# B&R Automation Studio project MappAssetInt
Automation Studio 4.12.6.106; technology packages: mapp 5.24.2

## Configuration X20CP

CPU X20CP3687X, AutomationRuntime J4.93, Build 4.1.2, Safety 0.0, Vc V4.73.3

### Task classes (Cpu.sw)
```
Cyclic#8:
  AssetTest <- AssetTest.prg
  Sample <- exAssetInt.Sample.prg
  Shift <- Shift.prg
VcDataObjects: Vis <- Vis.dob
Binaries: vcnet, udbdef, vcrt, vcpkat, vcctext, vctcal, vcfile, vcgclass, vccstr, vcpdsw, arial, vcdsint, vcmgr, vcdsloc, vcfntttf, vccovl, vcshared, arialbd, vcalarm, vccdt, vcpdvnc, vcpfar00, vcbclass, TCData, vccnum, arsvcreg, vccshape, vccbtn, vccddbox, Vis01, Vis02, Vis03, vcclbox, vccpopup, arconfig, User, Config, ashwd, ashwac, Role, asfw, iomap, sysconf, vcpfx20, Visu01, Visu03, Visu02, Config_1
Libraries: AsBrStr, MpData, MpBase, MpAssetInt, MpCom, FileIO, DataObj, astime, brsystem, sys_lib, runtime, standard, vcresman, asieccon, ashw, AsIODiag, exAssetInt
```

### Hardware
```
X20CP3687X : X20CP3687X v1.8.0.0
  Connector IF2:
    ActivateDevice = 1
    Vnc1
    VncVcObjectName1 = Vis
    VncKeyMappingFile1 = VC\PS2-Keyboard.dis
    VncRefreshRate1 = 500
    ActivateSnmp = 2
  Connector IF3:
    DNAConfiguration = manual
    CycleTime = 2000
  ConfigurationID = MappAssetInt_X20CP1583
  UserPartitionSize = 16
  Simulation = 1
  UserRamSize = 731936
  RemMemSize = 300000
  TimerDeviceType = EPLX2X
  TimerDevice = X20CP3687X.IF3
  TaskClassIdleTime = 2000
  Cyclic1Duration = 2000
  Cyclic8Stack = 20000
  FileDevice1
  FileDeviceName1 = ARsim
  FileDevicePath1 = C:\Temp\AssetInt
  FileDevice2
  FileDeviceName2 = USER_HD
  FileDevicePath2 = F:\
  FtpUser1
  FtpUsername1 = admin
  FtpUserPassword1 = WA9hSMBXiqkZliudaf2dLB8I5WaEURjKd6F9iexMfBQ=
  FtpUserSalt1 = wS51ak4d
  FTPAccessRight1 = 0
  ActivateOpcUa = 1
  OpcUaInformationModels_PV_Version = 1
```

### Config.mpassetintcore - X20CP3687X/mappServices/Config.mpassetintcore
```
Element gAssetIntCore (Type=mpassetintcore)
  AssetInt:
    Shifts:
      [0]:
        Name = Morning
        TotalTime:
          Start = 21600000
          End = 50400000
        ScheduledDowntime:
          [0]:
            Reason = Lunch
            Start = 21780000
            End = 21900000
      [1]:
        Name = Afternoon
        TotalTime:
          Start = 50400000
          End = 79200000
        ScheduledDowntime:
          [0]:
            Reason = Dinner
            Start = 64800000
            End = 66600000
      [2]:
        Name = Night
        TotalTime:
          Start = 79200000
          End = 21600000
    Export:
      ColumnSeparator = ;
      DecimalMark = ,
  Alarms = MpAlarmX
```

## Configuration X20CP1583

CPU X20CP3586, AutomationRuntime I4.93, Build 4.1.2, Safety 0.0, Vc V4.73.1

CPU X20CP3687X, AutomationRuntime I4.93, Build 4.1.2, Safety 0.0, Vc V4.73.1

### Task classes (Cpu.sw)
```
Cyclic#4:
  AssetTest <- AssetTest.prg
Cyclic#8:
  Sample <- exAssetInt.Sample.prg
  Shift <- Shift.prg
VcDataObjects: Visu_R <- Visu_Resized.dob
Binaries: vcnet, udbdef, vcrt, vcpkat, vcctext, Visu01, vctcal, Visu03, vcfile, vcgclass, vccstr, vcpdsw, arial, vcdsint, vcmgr, vcdsloc, vcfntttf, Visu02, vccovl, vcshared, arialbd, vcalarm, vccdt, vcpdvnc, vcpfar00, vcbclass, TCData, vccnum, arsvcreg, vccshape, vccbtn, arconfig, User, Config, ashwd, ashwac, Role, asfw, iomap, sysconf, vcpfx20, Config_1
Libraries: AsBrStr, MpData, MpBase, MpAssetInt, MpCom, FileIO, DataObj, astime, brsystem, sys_lib, runtime, exAssetInt, vcresman, asieccon, ashw, standard
```

### Hardware
```
X20CP3687X : X20CP3687X v1.8.0.0
  Connector IF2:
    ActivateDevice = 1
    Vnc1
    VncVcObjectName1 = Vis
    VncKeyMappingFile1 = VC\PS2-Keyboard.dis
    VncRefreshRate1 = 500
    ActivateSnmp = 2
  Connector IF3:
    DNAConfiguration = manual
    CycleTime = 2000
  ConfigurationID = MappAssetInt_X20CP1583
  UserPartitionSize = 16
  UserRamSize = 731936
  RemMemSize = 300000
  Cyclic8Stack = 20000
  FileDevice1
  FileDeviceName1 = ARsim
  FileDevicePath1 = c:\Temp\AssetInt
  FileDevice2
  FileDeviceName2 = USER_HD
  FileDevicePath2 = f:\
  FtpUser1
  FtpUsername1 = admin
  FtpUserPassword1 = WA9hSMBXiqkZliudaf2dLB8I5WaEURjKd6F9iexMfBQ=
  FtpUserSalt1 = wS51ak4d
  FTPAccessRight1 = 0
```

### Config.mpassetintcore - X20CP3586/mappServices/Config.mpassetintcore
```
Element gAssetIntCore (Type=mpassetintcore)
  AssetInt:
    Shifts:
      [0]:
        Name = Morning
        TotalTime:
          Start = 21600000
          End = 50400000
        ScheduledDowntime:
          [0]:
            Reason = Lunch
            Start = 39600000
            End = 41400000
      [1]:
        Name = Afternoon
        TotalTime:
          Start = 50400000
          End = 79200000
        ScheduledDowntime:
          [0]:
            Reason = Dinner
            Start = 64800000
            End = 66600000
      [2]:
        Name = Night
        TotalTime:
          Start = 79200000
          End = 21600000
    Export:
      ColumnSeparator = ;
      DecimalMark = ,
  Alarms = MpAlarmX
```

### Config_1.mpdatarecorder - X20CP3586/mappServices/Config_1.mpdatarecorder
```
Element gDataRecorder (Type=mpdatarecorder)
  DataRecorder:
    MaxFileSize = 2000
    SaveInterval = 3600000
    BufferSize = 70
    TimeStampPattern = %Y %m %d %H:%M:%S
    AutoSave = FALSE
    OverwriteOldestFile = TRUE
  Alarms = MpAlarmX
```

## Configuration X20EM

CPU X20EM0612, AutomationRuntime J4.93, Build 4.1.2, Safety 0.0, Vc V4.73.2

### Task classes (Cpu.sw)
```
Cyclic#8:
  AssetTest <- AssetTest.prg
  Sample <- exAssetInt.Sample.prg
  Shift <- Shift.prg
VcDataObjects: Vis <- Vis.dob
Binaries: vcnet, udbdef, vcrt, vcpkat, vcctext, vctcal, vcfile, vcgclass, vccstr, vcpdsw, arial, vcdsint, vcmgr, vcdsloc, vcfntttf, vccovl, vcshared, arialbd, vcalarm, vccdt, vcpdvnc, vcpfar00, vcbclass, TCData, vccnum, arsvcreg, vccshape, vccbtn, vccddbox, Vis01, Vis02, Vis03, vcclbox, vccpopup, arconfig, User, Config, ashwd, ashwac, Role, asfw, iomap, sysconf, vcpfx20, Visu01, Visu03, Visu02, Config_1
Libraries: AsBrStr, MpData, MpBase, MpAssetInt, MpCom, FileIO, DataObj, astime, brsystem, sys_lib, runtime, exAssetInt, standard, vcresman, asieccon, ashw, AsIODiag
```

### Hardware
```
X20EM0612 : X20EM0612 v1.1.1.0
  Connector IF2:
    ActivateDevice = 1
    Vnc1
    VncVcObjectName1 = Visu
    VncKeyMappingFile1 = VC\PS2-Keyboard.dis
    VncRefreshRate1 = 500
    ActivateSnmp = 2
  Connector IF3:
    DNAConfiguration = manual
  ConfigurationID = MappAssetInt_X20CP1583
  UserPartitionSize = 16
  UserRamSize = 32000
  RemMemSize = 32000
  TimerDeviceType = EPLX2X
  TimerDevice = X20EM0612.IF3
  TaskClassIdleTime = 2000
  Cyclic1Duration = 2000
  Cyclic8Stack = 20000
  FileDevice1
  FileDeviceName1 = ARsim
  FileDevicePath1 = c:\Temp\AssetInt
  FileDevice2
  FileDeviceName2 = USER_HD
  FileDevicePath2 = f:\
  FtpUser1
  FtpUsername1 = admin
  FtpUserPassword1 = WA9hSMBXiqkZliudaf2dLB8I5WaEURjKd6F9iexMfBQ=
  FtpUserSalt1 = wS51ak4d
  FTPAccessRight1 = 0
  ActivateOpcUa = 1
  OpcUaInformationModels_PV_Version = 1
```

### Config.mpassetintcore - X20EM0612/mappServices/Config.mpassetintcore
```
Element gAssetIntCore (Type=mpassetintcore)
  AssetInt:
    RecordingSizeShiftStatistics = 8
    RecordingSizeTimeline = 8
    RecordingSizeJobStatistics = 8
    Shifts:
      [0]:
        Name = Morning
        TotalTime:
          Start = 21600000
          End = 50400000
        ScheduledDowntime:
          [0]:
            Reason = Lunch
            Start = 21780000
            End = 21900000
      [1]:
        Name = Afternoon
        TotalTime:
          Start = 50400000
          End = 79200000
        ScheduledDowntime:
          [0]:
            Reason = Dinner
            Start = 64800000
            End = 66600000
      [2]:
        Name = Night
        TotalTime:
          Start = 79200000
          End = 21600000
    Export:
      ColumnSeparator = ;
      DecimalMark = ,
  Alarms = MpAlarmX
```

## Logical view

Binary libraries used (declarations not repeated): operator, runtime, astime, AsIecCon, sys_lib, DataObj, brsystem, FileIO, AsBrStr, standard, AsIODiag, MpAssetInt 5.24.2

### Global.typ - Globale Datentypen
```iecst
TYPE
	TIME_typ : 	STRUCT
		Hour : UDINT;
		Minutes : UDINT;
	END_STRUCT;
	SHIFT_typ : 	STRUCT
		Start : TIME_typ;
		End : TIME_typ;
		Name : STRING[20];
		ScheduledDowntime : ARRAY[0..9]OF DOWNTIME_typ;
	END_STRUCT;
	DOWNTIME_typ : 	STRUCT
		Start : TIME_typ;
		End : TIME_typ;
		Reason : STRING[20];
	END_STRUCT;
END_TYPE
```

### Global.var - Globale Variablen
```iecst
(*.-.-.-.-.---------------------------------------------------------------------------------------------------------------------------------------------------------------------------------*)
VAR
	gShift : ARRAY[0..4] OF SHIFT_typ;
	gAdditionalData : STRING[255] := 'Choclate';
	gNominalProductionRate : REAL := 3600;
	gDeviceName : STRING[50];
	gPieceCounterJob : UDINT;
	gPieceCounter : UDINT;
	gRejectCounter : UDINT;
	gRejectCounterRatio : UDINT := 10;
	gCurrentUser : STRING[50] := 'TylerDurden';
	gJobName : STRING[20] := 'Cookies';
	gDowntimeReason : STRING[50] := 'Winder is broken';
	gDowntime : exAssetIntDowntimeEnum;
	gCommandUpdate : BOOL;
	gCommandReset : BOOL;
	gCommandExport : BOOL;
	gCommandResetError : BOOL;
	gEnable : BOOL := TRUE;
	gLocked : UINT := 0;
END_VAR
```


### Program Logical/Shift (IEC)

#### Cyclic.st - Cyclic code
```iecst
PROGRAM _CYCLIC

	AssetIntPar.NominalProductionRate := gNominalProductionRate;
	AssetIntPar.AdditionalData := gAdditionalData;
	AssetIntPar.CurrentUser := gCurrentUser;
	AssetIntPar.Job := gJobName;

	MpAssetIntCore_0.PieceCounter := gPieceCounter;
	MpAssetIntCore_0.RejectCounter := gRejectCounter;

    MpAssetIntCore_0.MpLink := ADR(gAssetIntCore);
    MpAssetIntCore_0.Enable := gEnable;
    MpAssetIntCore_0.Parameters := ADR(AssetIntPar);
	MpAssetIntCore_0.DeviceName := ADR(gDeviceName);
	MpAssetIntCore_0.DowntimeReason := ADR(gDowntimeReason);
	MpAssetIntCore_0.Downtime := UDINT_TO_UINT(gDowntime);
	MpAssetIntCore_0.Update := gCommandUpdate;
	MpAssetIntCore_0.Reset := gCommandReset;
	MpAssetIntCore_0.Export := gCommandExport;
	MpAssetIntCore_0();

	IF EDGEPOS(MpAssetIntCore_0.UpdateDone) THEN
		gCommandUpdate := FALSE;
	END_IF

	AssetIntConfig.Export.DecimalMark := ',';
	AssetIntConfig.Export.ColumnSeparator := ';';
    brsstrcpy(ADR(AssetIntConfig.Export.JobStatisticsFileNamePattern), ADR('1234JobStatistics_%Y_%m_%d_%H_%M.csv'));
    brsstrcpy(ADR(AssetIntConfig.Export.ShiftStatisticsFileNamePattern), ADR('1234ShiftStatistics_%Y_%m_%d_%H_%M.csv'));
    brsstrcpy(ADR(AssetIntConfig.Export.TimelineFileNamePattern), ADR('1234Timeline_%Y_%m_%d_%H_%M.csv'));

	// --------------------------------------------------------------------------------------------------------------------------
	// Asset configuration
	FOR x := 0 TO SIZEOF(AssetIntConfig.Shifts)/SIZEOF(AssetIntConfig.Shifts[0]) - 1 DO
		AssetIntConfig.Shifts[x].Name := gShift[x].Name;
		FOR y := 0 TO SIZEOF(AssetIntConfig.Shifts[x].ScheduledDowntime)/SIZEOF(AssetIntConfig.Shifts[x].ScheduledDowntime[0]) - 1 DO
			AssetIntConfig.Shifts[x].ScheduledDowntime[y].Reason := gShift[x].ScheduledDowntime[y].Reason;
			AssetIntConfig.Shifts[x].ScheduledDowntime[y].Start := UDINT_TO_TOD((gShift[x].ScheduledDowntime[y].Start.Hour * 3600000) + (gShift[x].ScheduledDowntime[y].Start.Minutes * 60000));
			AssetIntConfig.Shifts[x].ScheduledDowntime[y].End := UDINT_TO_TOD((gShift[x].ScheduledDowntime[y].End.Hour * 3600000) + (gShift[x].ScheduledDowntime[y].End.Minutes * 60000));
		END_FOR;
		AssetIntConfig.Shifts[x].TotalTime.Start := UDINT_TO_TOD((gShift[x].Start.Hour * 3600000) + (gShift[x].Start.Minutes * 60000));
		AssetIntConfig.Shifts[x].TotalTime.End := UDINT_TO_TOD((gShift[x].End.Hour * 3600000) + (gShift[x].End.Minutes * 60000));
	END_FOR;

	IF (AssetIntConfig.Shifts[1].TotalTime.Start = AssetIntConfig.Shifts[0].TotalTime.End) AND (AssetIntConfig.Shifts[1].TotalTime.End <> AssetIntConfig.Shifts[1].TotalTime.Start) THEN
		AssetIntConfig.Shifts[1].TotalTime.Start := UDINT_TO_TOD((gShift[1].Start.Hour * 3600000) + (gShift[1].Start.Minutes * 60000) + 1);
	END_IF

	IF (AssetIntConfig.Shifts[2].TotalTime.Start = AssetIntConfig.Shifts[1].TotalTime.End) AND (AssetIntConfig.Shifts[2].TotalTime.End <> AssetIntConfig.Shifts[2].TotalTime.Start)  THEN
		AssetIntConfig.Shifts[2].TotalTime.Start := UDINT_TO_TOD((gShift[2].Start.Hour * 3600000) + (gShift[2].Start.Minutes * 60000) + 1);
	END_IF

	IF (AssetIntConfig.Shifts[0].TotalTime.Start = AssetIntConfig.Shifts[2].TotalTime.End) THEN
		AssetIntConfig.Shifts[0].TotalTime.Start := UDINT_TO_TOD((gShift[0].Start.Hour * 3600000) + (gShift[0].Start.Minutes * 60000) + 1);
	END_IF

    IF (AssetIntConfig.Shifts[1].TotalTime.Start = AssetIntConfig.Shifts[0].TotalTime.End) AND (AssetIntConfig.Shifts[1].TotalTime.End <> AssetIntConfig.Shifts[1].TotalTime.Start) THEN
        AssetIntConfig.Shifts[1].TotalTime.Start := UDINT_TO_TOD((gShift[1].Start.Hour * 3600000) + (gShift[1].Start.Minutes * 60000) + 1);
    END_IF

    IF (AssetIntConfig.Shifts[2].TotalTime.Start = AssetIntConfig.Shifts[1].TotalTime.End) AND (AssetIntConfig.Shifts[2].TotalTime.End <> AssetIntConfig.Shifts[2].TotalTime.Start)  THEN
        AssetIntConfig.Shifts[2].TotalTime.Start := UDINT_TO_TOD((gShift[2].Start.Hour * 3600000) + (gShift[2].Start.Minutes * 60000) + 1);
    END_IF

    IF (AssetIntConfig.Shifts[0].TotalTime.Start = AssetIntConfig.Shifts[2].TotalTime.End) THEN
        AssetIntConfig.Shifts[0].TotalTime.Start := UDINT_TO_TOD((gShift[0].Start.Hour * 3600000) + (gShift[0].Start.Minutes * 60000) + 1);
    END_IF

    IF (MpAssetIntCoreConfig_0.Save = 1) AND (MpAssetIntCoreConfig_0.CommandDone = 1) AND (MpAssetIntCoreConfig_0.CommandBusy = 0) THEN
        MpAssetIntCoreConfig_0.Save := 0;
    END_IF

    MpAssetIntCoreConfig_0.MpLink :=  ADR(gAssetIntCore);
    MpAssetIntCoreConfig_0.Enable := MpAssetIntCore_0.Active AND NOT DisableConfig;
    MpAssetIntCoreConfig_0.Configuration := ADR(AssetIntConfig);
    MpAssetIntCoreConfig_0();

    MpAssetIntShiftListUI_0.MpLink :=  ADR(gAssetIntCore);
    MpAssetIntShiftListUI_0.Enable := MpAssetIntCore_0.Active;
    MpAssetIntShiftListUI_0.UIConnect := ADR(ShiftListUIConnect);
	MpAssetIntShiftListUI_0.UISetup := ShiftListUISetup;
	MpAssetIntShiftListUI_0();

    MpAssetIntJobListUI_0.MpLink :=  ADR(gAssetIntCore);
    MpAssetIntJobListUI_0.Enable := MpAssetIntCore_0.Active;
	MpAssetIntJobListUI_0.UIConnect := ADR(JobListUIConnect);
	MpAssetIntJobListUI_0.UISetup := JobListUISetup;
	MpAssetIntJobListUI_0();

	MpAssetIntTimelineUI_0.MpLink :=  ADR(gAssetIntCore);
	MpAssetIntTimelineUI_0.Enable := MpAssetIntCore_0.Active;
	MpAssetIntTimelineUI_0.UIConnect := ADR(TimelineUIConnect);
	MpAssetIntTimelineUI_0.UISetup := TimelineUISetup;
	MpAssetIntTimelineUI_0();

END_PROGRAM
```

#### Init.st - Init code
```iecst
PROGRAM _INIT
	MpAssetIntCoreConfig_0.Save := TRUE;
END_PROGRAM
```

#### Exit.st - Exit code
```iecst
(*********************************************************************************
 * Copyright: Bernecker + Rainer
 * Author:    heinesm
 * Created:   11. August 2017/14:15
 *********************************************************************************)
PROGRAM _EXIT
MpAssetIntCore_0.Enable := 0;
MpAssetIntCore_0();
MpAssetIntCoreConfig_0.Enable := 0;
MpAssetIntCoreConfig_0();
MpAssetIntShiftListUI_0.Enable := 0;
MpAssetIntShiftListUI_0();
MpAssetIntJobListUI_0.Enable := 0;
MpAssetIntJobListUI_0();
END_PROGRAM
```

#### Variables.var - Local variables
```iecst
VAR
	y : USINT;
	x : USINT;
	DisableConfig : BOOL;
	MpAssetIntCore_0 : MpAssetIntCore;
	AssetIntPar : MpAssetIntParType;
	MpAssetIntCoreConfig_0 : MpAssetIntCoreConfig;
	AssetIntConfig : MpAssetIntCoreConfigType;
	MpAssetIntShiftListUI_0 : MpAssetIntShiftListUI;
	MpAssetIntJobListUI_0 : MpAssetIntJobListUI;
	MpAssetIntTimelineUI_0 : MpAssetIntTimelineUI;
	JobListUIConnect : MpAssetIntJobListUIConnectType;
	ShiftListUIConnect : MpAssetIntShiftListUIConnectType;
	TimelineUIConnect : MpAssetIntTimelineUIConnectType;
	ShiftListUISetup : MpAssetIntShiftListUISetupType;
	TimelineUISetup : MpAssetIntTimelineUISetupType;
	JobListUISetup : MpAssetIntJobListUISetupType := (OutputListSize:=8,ScrollWindow:=2);
END_VAR
```

### Program Logical/AssetTest (IEC)

#### Main.st - Init, cyclic, exit code
```iecst
PROGRAM _INIT
	PV_xgetadr(ADR('Sample:exAssetIntCore_0'), ADR(exAssetIntCoreAdr), ADR(exAssetIntCoreLen));
	exAssetIntCore_0 ACCESS exAssetIntCoreAdr;

END_PROGRAM

PROGRAM _CYCLIC
	// Count time it takes the function block to become active
	IF exAssetIntCore_0.Enable = TRUE AND exAssetIntCore_0.Active = FALSE THEN
		TestBootCounter := TestBootCounter + 1;
	END_IF

	// Get current date and time
	IF GetDateTime THEN
		RTC_gettime(ADR(RTCtime_struct));
		GetDateTime := FALSE;
	END_IF

	// Set current date and time
	IF SetDateTime THEN
		RTC_settime(ADR(RTCtime_struct));
		SetDateTime := FALSE;
	END_IF

	// Auto count pieces
	IF AutoCount THEN
		AutoCountTime.IN := TRUE;
		AutoCountTime.PT := AutoCountCycle / 10;
		AutoCountTime();

		IF AutoCountTime.Q THEN
			AutoCountTime.IN := FALSE;
			AutoCountTime();

			gPieceCounter := gPieceCounter + 1;

			// Generate reject parts
			IF gPieceCounter MOD gRejectCounterRatio = 0 THEN
				gRejectCounter := gRejectCounter + 1;
			END_IF
		END_IF
	END_IF

	// Create new jobs
	IF AutoCreateJobs THEN
		AutoCount := TRUE;

		IF gPieceCounter > AutoCreatePieceCnt + AutoCreateJobsNum THEN
			AutoCreatePieceCnt := gPieceCounter;
			AutoCreateJobsCnt := AutoCreateJobsCnt + 1;

			// Create new job name
			TmpStr1 := 'Job';
			brsitoa(AutoCreateJobsCnt, ADR(TmpStr2));
			brsstrcat(ADR(TmpStr1), ADR(TmpStr2));
			gJobName := TmpStr1;
			gCommandUpdate := TRUE;

		END_IF

	END_IF

	// Copy internal memory buffer to structure for debugging
//	IF exAssetIntLink.Memory <> 0 THEN
//		brsmemcpy(ADR(Memory), exAssetIntLink.Memory, SIZEOF(Memory));
//	ELSE
//		brsmemset(ADR(Memory), 0, SIZEOF(Memory));
//	END_IF

	TestCase1;
	TestCase2;
END_PROGRAM
```

#### Types.typ - Local data types
```iecst
TYPE
	TestResultEnum :
		(
		TestResultWaiting,
		TestResultRunning,
		TestResultPassed,
		TestResultFailed
		);
END_TYPE
```

#### Variables.var - Local variables
```iecst
(*.-.-.-.-.---------------------------------------------------------------------------------------------------------------------------------------------------------------------------------*)
VAR
	Memory : ARRAY[0..19] OF exCoreInternalRecordType;
	TmpStr1 : STRING[80];
	TmpStr2 : STRING[80];
END_VAR
(*.-.-.-.-.---------------------------------------------------------------------------------------------------------------------------------------------------------------------------------*)
VAR
	AutoCount : BOOL; (*Start auto count*)
END_VAR
VAR CONSTANT
	AutoCountCycle : UINT := 1000; (*Auto count cycle in ms*)
END_VAR
VAR
	AutoCountTime : TON_10ms;
END_VAR
(*.-.-.-.-.---------------------------------------------------------------------------------------------------------------------------------------------------------------------------------*)
VAR
	AutoCreateJobs : BOOL; (*Auto create jobs*)
	AutoCreatePieceCnt : UDINT; (*Job piece counter*)
	AutoCreateJobsCnt : UDINT; (*Job name counter*)
END_VAR
VAR CONSTANT
	AutoCreateJobsNum : UDINT := 30; (*Pieces per job auto create*)
END_VAR
(*.-.-.-.-.---------------------------------------------------------------------------------------------------------------------------------------------------------------------------------*)
VAR
	GetDateTime : BOOL;
	SetDateTime : BOOL;
	RTCtime_struct : RTCtime_typ;
END_VAR
(*.-.-.-.-.---------------------------------------------------------------------------------------------------------------------------------------------------------------------------------*)
VAR
	TestBootCounter : UDINT;
	TestResult : ARRAY[1..9] OF TestResultEnum;
	TestCase : ARRAY[1..9] OF BOOL;
	TestState : ARRAY[1..9] OF USINT;
	TestIdle : ARRAY[1..9] OF UDINT;
	TesMyId : USINT;
END_VAR
(*.-.-.-.-.---------------------------------------------------------------------------------------------------------------------------------------------------------------------------------*)
VAR
	exAssetIntCoreAdr : {REDUND_UNREPLICABLE} UDINT;
	exAssetIntCoreLen : {REDUND_UNREPLICABLE} UDINT;
	exAssetIntCore_0 : REFERENCE TO exAssetIntCore;
END_VAR
```

#### TestCase1.st
```iecst
// What is this test case doing?
// 1. Set PLC time to first shift end minus 2 minutes
// 2. Wait 5 minutes for shift to change
// 3. Set PLC time to second shift end minus 2 minutes
// 4. Wait 5 minutes for shift to change
// 5. Set PLC time to third shift end minus 2 minutes
// 6. Wait 5 minutes for shift to change
//
// What is this test case testing?
// Make sure shift changeover is handled correct
// Make sure gaps in shifts are handled correct
//
// What should be the preset?
// At least 3 shifts, a gap between one shift end and the next shift start

ACTION TestCase1:
	TesMyId := 1;
	IF TestCase[1] THEN
		CASE TestState[TesMyId] OF
			0:
				AutoCount := TRUE;
				RTC_gettime(ADR(RTCtime_struct));
				TestIdle[TesMyId] := 0;

				TestState[TesMyId] := TestState[TesMyId] + 1;
			1:
				IF gShift[0].End.Minutes > 5 THEN
					RTCtime_struct.hour := UDINT_TO_USINT(gShift[0].End.Hour);
					RTCtime_struct.minute := UDINT_TO_USINT(gShift[0].End.Minutes)-2;
				ELSE
					RTCtime_struct.hour := UDINT_TO_USINT(gShift[0].End.Hour)-1;
					RTCtime_struct.minute := 58;
				END_IF
				RTC_settime(ADR(RTCtime_struct));

				TestState[TesMyId] := TestState[TesMyId] + 1;
			2:
				TestIdle[TesMyId] := TestIdle[TesMyId] + 1;
				IF TestIdle[TesMyId] > 100*60*5 THEN
					TestIdle[TesMyId] := 0;
					TestState[TesMyId] := TestState[TesMyId] + 1;
				END_IF
			3:
				IF gShift[1].End.Minutes > 5 THEN
					RTCtime_struct.hour := UDINT_TO_USINT(gShift[1].End.Hour);
					RTCtime_struct.minute := UDINT_TO_USINT(gShift[1].End.Minutes)-2;
				ELSE
					RTCtime_struct.hour := UDINT_TO_USINT(gShift[1].End.Hour)-1;
					RTCtime_struct.minute := 58;
				END_IF
				RTC_settime(ADR(RTCtime_struct));

				TestState[TesMyId] := TestState[TesMyId] + 1;
			4:
				TestIdle[TesMyId] := TestIdle[TesMyId] + 1;
				IF TestIdle[TesMyId] > 100*60*5 THEN
					TestIdle[TesMyId] := 0;
					TestState[TesMyId] := TestState[TesMyId] + 1;
				END_IF
			5:
				IF gShift[2].End.Minutes > 5 THEN
					RTCtime_struct.hour := UDINT_TO_USINT(gShift[2].End.Hour);
					RTCtime_struct.minute := UDINT_TO_USINT(gShift[2].End.Minutes)-2;
				ELSE
					RTCtime_struct.hour := UDINT_TO_USINT(gShift[2].End.Hour)-1;
					RTCtime_struct.minute := 58;
				END_IF
				RTC_settime(ADR(RTCtime_struct));

				TestState[TesMyId] := TestState[TesMyId] + 1;
			6:
				TestIdle[TesMyId] := TestIdle[TesMyId] + 1;
				IF TestIdle[TesMyId] > 100*60*5 THEN
					TestCase[TesMyId] := FALSE;
					TestState[TesMyId] := 0;
				END_IF
		END_CASE;
	END_IF
END_ACTION
```

#### TestCase2.st
```iecst
// What is this test case doing?
// 1. Set 3 scheduled downtimes for first shift
// 1. Set PLC time to first shift start
// 2. Wait 20 minutes for shift to change
//
// What is this test case testing?
// Make sure preconfigured scheduled downtime is handled correct
//
// What should be the preset?
// At least 1 shift

ACTION TestCase2:
	TesMyId := 2;
	IF TestCase[TesMyId] THEN
		CASE TestState[TesMyId] OF
			0:
				TestResult[TesMyId] := TestResultRunning;
				AutoCount := TRUE;
				RTC_gettime(ADR(RTCtime_struct));
				TestIdle[TesMyId] := 0;

				TestState[TesMyId] := TestState[TesMyId] + 1;
			1:
				gShift[0].ScheduledDowntime[0].Start.Hour := gShift[0].Start.Hour;
				gShift[0].ScheduledDowntime[0].Start.Minutes := gShift[0].Start.Minutes + 3;
				gShift[0].ScheduledDowntime[0].End.Hour := gShift[0].Start.Hour;
				gShift[0].ScheduledDowntime[0].End.Minutes := gShift[0].Start.Minutes + 5;
				gShift[0].ScheduledDowntime[0].Reason := 'Test Reason 1';

				gShift[0].ScheduledDowntime[1].Start.Hour := gShift[0].Start.Hour;
				gShift[0].ScheduledDowntime[1].Start.Minutes := gShift[0].Start.Minutes + 3;
				gShift[0].ScheduledDowntime[1].End.Hour := gShift[0].Start.Hour;
				gShift[0].ScheduledDowntime[1].End.Minutes := gShift[0].Start.Minutes + 5;
				gShift[0].ScheduledDowntime[1].Reason := 'Test Reason 2';

				gShift[0].ScheduledDowntime[2].Start.Hour := gShift[0].Start.Hour;
				gShift[0].ScheduledDowntime[2].Start.Minutes := gShift[0].Start.Minutes + 3;
				gShift[0].ScheduledDowntime[2].End.Hour := gShift[0].Start.Hour;
				gShift[0].ScheduledDowntime[2].End.Minutes := gShift[0].Start.Minutes + 5;
				gShift[0].ScheduledDowntime[2].Reason := 'Test Reason 3';

				RTCtime_struct.hour := UDINT_TO_USINT(gShift[0].Start.Hour);
				RTCtime_struct.minute := UDINT_TO_USINT(gShift[0].Start.Minutes);
				RTC_settime(ADR(RTCtime_struct));

				TestState[TesMyId] := TestState[TesMyId] + 1;
			2:
				TestIdle[TesMyId] := TestIdle[TesMyId] + 1;
				IF TestIdle[TesMyId] > 100*60*17 THEN
					TestIdle[TesMyId] := 0;
					TestState[TesMyId] := TestState[TesMyId] + 1;
				END_IF
			3:
				TestCase[TesMyId] := FALSE;
				TestState[TesMyId] := 0;
				IF exAssetIntCore_0.Info.ShiftStatistics.ScheduledDowntime.Minutes = 6 THEN
					TestResult[TesMyId] := TestResultPassed;
				ELSE
					TestResult[TesMyId] := TestResultFailed;
				END_IF
		END_CASE;
	END_IF
END_ACTION
```

### Program Logical/exAssetInt/Sample (IEC)

#### Variables.var
```iecst
(*Remanet cross link variable*)
VAR RETAIN
	exAssetIntLink : exAssetIntLinkType;
END_VAR
(*Asset core*)
VAR
	exAssetIntCore_0 : exAssetIntCore;
	exAssetIntPar : exAssetIntParType;
	LoggerCore : ARRAY[0..LOG_NUM] OF STRING[LOG_LEN];
END_VAR
(*Asset configuration*)
VAR
	exAssetIntConfig_0 : exAssetIntCoreConfig;
	exAssetIntConfig : exAssetIntCoreConfigType;
	LoggerConfig : ARRAY[0..LOG_NUM] OF STRING[LOG_LEN];
END_VAR
(*Asset UI function blocks*)
VAR
	exAssetIntJobListUI_0 : exAssetIntJobListUI;
	JobListUIConnect : exAssetIntJobListUIConnectType;
	LoggerUIJob : ARRAY[0..LOG_NUM] OF STRING[LOG_LEN];
	exAssetIntShiftListUI_0 : exAssetIntShiftListUI;
	ShiftListUIConnect : exAssetIntShiftListUIConnectType;
	LoggerUIShift : ARRAY[0..LOG_NUM] OF STRING[LOG_LEN];
	exAssetIntTimelineUI_0 : exAssetIntTimelineUI;
	TimelineUIConnect : exAssetIntTimelineUIConnectType;
	LoggerUITimeline : ARRAY[0..LOG_NUM] OF STRING[LOG_LEN];
	y : USINT;
	x : USINT;
END_VAR
```

#### Cyclic.st
```iecst
PROGRAM _CYCLIC
	// --------------------------------------------------------------------------------------------------------------------------
	// Asset configuration
	FOR x := 0 TO SIZEOF(exAssetIntConfig.Shifts)/SIZEOF(exAssetIntConfig.Shifts[0]) - 1 DO
		exAssetIntConfig.Shifts[x].Name := gShift[x].Name;
		FOR y := 0 TO SIZEOF(exAssetIntConfig.Shifts[x].ScheduledDowntime)/SIZEOF(exAssetIntConfig.Shifts[x].ScheduledDowntime[0]) - 1 DO
			exAssetIntConfig.Shifts[x].ScheduledDowntime[y].Reason := gShift[x].ScheduledDowntime[y].Reason;
			exAssetIntConfig.Shifts[x].ScheduledDowntime[y].Start := UDINT_TO_TOD((gShift[x].ScheduledDowntime[y].Start.Hour * 3600000) + (gShift[x].ScheduledDowntime[y].Start.Minutes * 60000));
			exAssetIntConfig.Shifts[x].ScheduledDowntime[y].End := UDINT_TO_TOD((gShift[x].ScheduledDowntime[y].End.Hour * 3600000) + (gShift[x].ScheduledDowntime[y].End.Minutes * 60000));
		END_FOR;
		exAssetIntConfig.Shifts[x].TotalTime.Start := UDINT_TO_TOD((gShift[x].Start.Hour * 3600000) + (gShift[x].Start.Minutes * 60000));
		exAssetIntConfig.Shifts[x].TotalTime.End := UDINT_TO_TOD((gShift[x].End.Hour * 3600000) + (gShift[x].End.Minutes * 60000));
	END_FOR;

	exAssetIntConfig_0.Enable := exAssetIntCore_0.Active;
	exAssetIntConfig_0.exLink := ADR(exAssetIntLink);
	exAssetIntConfig_0.DeviceName := ADR(gDeviceName);
	exAssetIntConfig_0.Configuration := ADR(exAssetIntConfig);
	exAssetIntConfig_0.Logger := ADR(LoggerConfig);
	exAssetIntConfig_0();

	// --------------------------------------------------------------------------------------------------------------------------
	// Transfer global parameters
	exAssetIntPar.NominalProductionRate := gNominalProductionRate;
	exAssetIntPar.AdditionalData := gAdditionalData;
	exAssetIntPar.CurrentUser := gCurrentUser;
	exAssetIntPar.Job := gJobName;

	exAssetIntCore_0.Enable := gEnable;
	exAssetIntCore_0.exLink := ADR(exAssetIntLink);
	exAssetIntCore_0.Parameters := ADR(exAssetIntPar);
	exAssetIntCore_0.Configuration := ADR(exAssetIntConfig);
	exAssetIntCore_0.DeviceName := ADR(gDeviceName);
	exAssetIntCore_0.StorageName := ADR(gDeviceName);
	exAssetIntCore_0.DowntimeReason := ADR(gDowntimeReason);
	exAssetIntCore_0.Downtime := gDowntime;
	exAssetIntCore_0.PieceCounter := gPieceCounter;
	exAssetIntCore_0.RejectCounter := gRejectCounter;
	exAssetIntCore_0.Logger := ADR(LoggerCore);
	exAssetIntCore_0.Update := gCommandUpdate;
	exAssetIntCore_0.Reset := gCommandReset;
	exAssetIntCore_0.Export := gCommandExport;
	exAssetIntCore_0.ErrorReset := gCommandResetError;
	exAssetIntCore_0();

	IF EDGEPOS(exAssetIntCore_0.UpdateDone) THEN
		gCommandUpdate := FALSE;
	END_IF

	// --------------------------------------------------------------------------------------------------------------------------
	// UI function blocks
	exAssetIntJobListUI_0.Enable := exAssetIntCore_0.Active;
	exAssetIntJobListUI_0.exLink := ADR(exAssetIntLink);
	exAssetIntJobListUI_0.UIConnect := ADR(JobListUIConnect);
	exAssetIntJobListUI_0.Logger := ADR(LoggerUIJob);
	exAssetIntJobListUI_0();

	exAssetIntShiftListUI_0.Enable := exAssetIntCore_0.Active;
	exAssetIntShiftListUI_0.exLink := ADR(exAssetIntLink);
	exAssetIntShiftListUI_0.UIConnect := ADR(ShiftListUIConnect);
	exAssetIntShiftListUI_0.Logger := ADR(LoggerUIShift);
	exAssetIntShiftListUI_0();

	exAssetIntTimelineUI_0.Enable := exAssetIntCore_0.Active;
	exAssetIntTimelineUI_0.exLink :=  ADR(exAssetIntLink);
	exAssetIntTimelineUI_0.UIConnect := ADR(TimelineUIConnect);
	exAssetIntTimelineUI_0.Logger := ADR(LoggerUITimeline);
	exAssetIntTimelineUI_0();

END_PROGRAM
```

#### Init.st
```iecst
PROGRAM _INIT
	gLocked;					// VC helper

	// --------------------------------------------------------------------------------------------------------------------------
	// Shift configuration
	gShift[0].Name := 'Morning';
	gShift[0].Start.Hour := 8;
	gShift[0].Start.Minutes := 0;
	gShift[0].End.Hour := 14;
	gShift[0].End.Minutes := 0;
	gShift[0].ScheduledDowntime[0].Reason := 'Breakfast';
	gShift[0].ScheduledDowntime[0].Start.Hour := 9;
	gShift[0].ScheduledDowntime[0].End.Hour := 9;
	gShift[0].ScheduledDowntime[0].End.Minutes := 15;

	gShift[1].Name := 'Afternoon';
	gShift[1].Start.Hour := 14;
	gShift[1].Start.Minutes := 0;
	gShift[1].End.Hour := 22;
	gShift[1].End.Minutes := 0;

	gShift[2].Name := 'Night';
	gShift[2].Start.Hour := 22;
	gShift[2].Start.Minutes := 0;
	gShift[2].End.Hour := 8;
	gShift[2].End.Minutes := 0;

	// --------------------------------------------------------------------------------------------------------------------------
	// Export configuration
	exAssetIntConfig.Export.DecimalMark := ',';
	exAssetIntConfig.Export.ColumnSeparator := ';';

	exAssetIntConfig.Export.ShiftStatistics := TRUE;
	exAssetIntConfig.Export.ShiftStatisticsFileNamePattern := 'ShiftStatistics_%Y_%m_%d_%H_%M.csv';

	exAssetIntConfig.Export.JobStatistics := TRUE;
	exAssetIntConfig.Export.JobStatisticsFileNamePattern := 'JobStatistics_%Y_%m_%d_%H_%M.csv';

	exAssetIntConfig.Export.Timeline := TRUE;
	exAssetIntConfig.Export.TimelineFileNamePattern := 'Timeline_%Y_%m_%d_%H_%M.csv';

	// Check if we are running in simuulation
	IF DiagCpuIsARsim() THEN
		gDeviceName := 'ARsim';
	ELSE
		gDeviceName := 'USER_HD';
	END_IF
END_PROGRAM
```

### Library Logical/exAssetInt/exAssetInt (IEC, version 1.20.0)

#### exAssetIntError.typ
```iecst
(*File Version 1000*)
(*------------------------------------------------------------------------------------------------------------------------------------------------------------------------------------------------------------------------------------------------------------------------------------------------------------------------------------------------------*)

TYPE
	exAssetIntErrorEnum :
		( (* Error numbers of library exAssetInt *)
		exASSETINT_NO_ERROR := 0, (* No error *)
		exASSETINT_ERR_ACTIVATION := -1064239103, (* Could not create coexonent [Error: 1, 0xc0910001] *)
		exASSETINT_ERR_exLINK_NULL := -1064239102, (* exLink is NULL pointer [Error: 2, 0xc0910002] *)
		exASSETINT_ERR_exLINK_INVALID := -1064239101, (* exLink connection not allowed [Error: 3, 0xc0910003] *)
		exASSETINT_ERR_exLINK_CHANGED := -1064239100, (* exLink modified [Error: 4, 0xc0910004] *)
		exASSETINT_ERR_exLINK_CORRUPT := -1064239099, (* Invalid exLink contents [Error: 5, 0xc0910005] *)
		exASSETINT_ERR_exLINK_IN_USE := -1064239098, (* exLink already in use [Error: 6, 0xc0910006] *)
		exASSETINT_ERR_PAR_NULL := -1064239097, (* Parameters structure is a null pointer [Error: 7, 0xc0910007] *)
		exASSETINT_ERR_CONFIG_NULL := -1064239096, (* Configuration structure is null pointer [Error: 8, 0xc0910008] *)
		exASSETINT_ERR_CONFIG_NO_PV := -1064239095, (* Configuration pointer not PV [Error: 9, 0xc0910009] *)
		exASSETINT_ERR_CONFIG_LOAD := -1064239094, (* Error loading configuration {2:ConfigName} (ErrorCause: {1:ErrorNumber}) [Error: 10, 0xc091000a] *)
		exASSETINT_WRN_CONFIG_LOAD := -2137980917, (* Warning loading configuration [Warning: 11, 0x8091000b] *)
		exASSETINT_ERR_CONFIG_SAVE := -1064239092, (* Error saving configuration {2:ConfigName} (ErrorCause: {1:ErrorNumber}) [Error: 12, 0xc091000c] *)
		exASSETINT_ERR_CONFIG_INVALID := -1064239091, (* Invalid Configuration [Error: 13, 0xc091000d] *)
		exASSETINT_ERR_BUFFER_CREATE := -1064136704, (* Could not allocate memory (ErrorCause: {1:ErrorNumber}) [Error: 36864, 0xc0929000] *)
		exASSETINT_ERR_WRITE_EXPORT_FILE := -1064136703, (* Error writing export-file {2:FileName} at {3:DeviceName} (ErrorCause: {1:ErrorNumber}) [Error: 36865, 0xc0929001] *)
		exASSETINT_ERR_READ_BUFFER_ENTRY := -1064136702, (* Error reading event entries from {2:BufferName} (ErrorCause: {1:ErrorNumber}) [Error: 36866, 0xc0929002] *)
		exASSETINT_ERR_INVALID_FILE_DEV := -1064136701, (* Invalid file-device [Error: 36867, 0xc0929003] *)
		exASSETINT_ERR_MISSING_UICONNECT := -1064136700, (* Missing value on UIConnect [Error: 36868, 0xc0929004] *)
		exASSETINT_INF_WAIT_CORE_FB := 1083346949, (* Core is not active [Informational: 36869, 0x40929005] *)
		exASSETINT_ERR_EVENT_RECORDER := -1064136698, (* Event not recorded (ErrorCause: {1:ErrorNumber}) [Error: 36870, 0xc0929006] *)
		exASSETINT_ERR_INVALID_SHIFT := -1064136697, (* Invalid shift {2:ShiftName} in configuration: {3:Cause} [Error: 36871, 0xc0929007] *)
		exASSETINT_ERR_BUFFER_RESET := -1064136696 (* Could not reset buffer {2:BufferName} (ErrorCause: {1:ErrorNumber}) [Error: 36872, 0xc0929008] *)
		);
END_TYPE
```

#### exAssetIntAlarm.typ
```iecst
(*File Version 1000*)
(*------------------------------------------------------------------------------------------------------------------------------------------------------------------------------------------------------------------------------------------------------------------------------------------------------------------------------------------------------*)

TYPE
	exAssetIntCoreAlarmEnum :
		( (* Alarms of exAssetInt Core *)
		exASSETINT_ALM_EXPORT_STATISTICS := 0, (* Export shift statistics failed. *)
		exASSETINT_ALM_EXPORT_TIMELINE := 1, (* Export timeline failed. *)
		exASSETINT_ALM_EXPORT_JOB := 2, (* Export job statistics failed. *)
		exASSETINT_ALM_UNSCH_DOWNTIME := 3 (* Machine is in an unscheduled downtime phase *)
		);
END_TYPE
```

#### MpAssetInt.typ
```iecst
(*File Version 1007*)
(*------------------------------------------------------------------------------------------------------------------------------------------------------------------------------------------------------------------------------------------------------------------------------------------------------------------------------------------------------*)
(*Internal type*)

TYPE
	exCoreInternalDataType : 	STRUCT
		RecordIndexUsed : ARRAY[0..CORE_EVENT_NUM_MAX]OF BOOL; (*Next record ID*)
		RecordIndex : UINT; (*Next record ID*)
		RecordData : exCoreInternalRecordType;
		State : exAssetIntStateEnum;
		StateError : exAssetIntStateEnum := exASSETINT_STATE_NONE;
		InitAfterBoot : BOOL;
		TimeLastCallShift : TIME;
		DiffLastCallShift : UDINT;
		TimeLastCallProduction : TIME;
		DiffLastCallProduction : UDINT;
		JobPieceCounterOld : UDINT;
		JobRejectCounterOld : UDINT;
		ShiftPieceCounterOld : UDINT;
		ShiftRejectCounterOld : UDINT;
		ShiftId : SINT;
		ShiftName : STRING[20];
		TmpStr1 : STRING[500];
		TmpStr2 : STRING[50];
		Downtime : exAssetIntDowntimeEnum;
		DowntimeReason : STRING[50];
		ProductionTotalTime : UDINT;
		CurrentTime : DTGetTime;
		PowerOffTime : DATE_AND_TIME;
		TimeOfDay : TIME_OF_DAY;
		ShiftTotalTimeStart : UDINT;
		StatsRefresh : TON_10ms;
		BackupTimer : TON_10ms;
		DirCreate_0 : DirCreate;
		CreateMemory : CreateMemory;
		ReadEventData : ReadEventData;
		WriteEventData : WriteEventData;
		ReadLinkData : ReadLinkData;
		WriteLinkData : WriteLinkData;
		ExportEventData : ExportEventData;
		x : UINT;
		y : UINT;
	END_STRUCT;
	exCoreInternalRecordType : 	STRUCT
		CRC : USINT;
		FileName : STRING[80]; (*ID of the event*)
		EventType : exCoreInternalRecordEnum;
		TimeStart : DATE_AND_TIME; (*Event start*)
		TimeEnd : DATE_AND_TIME; (*Event end*)
		ShiftName : STRING[20]; (*Shift name*)
		JobName : STRING[20]; (*Job name.*)
		TotalTime : exAssetIntTimeType; (*Total time since this job started*)
		ScheduledDowntime : exAssetIntTimeType; (*Scheduled downtime since this job started*)
		UnscheduledDowntime : exAssetIntTimeType; (*Unsheduled downtime since this job started*)
		Uptime : exAssetIntTimeType; (*Uptime since this job started*)
		NominalProductionTime : exAssetIntTimeType; (*Time of production at nominal speed since this job started*)
		GoodProductionTime : exAssetIntTimeType; (*Time of good production since this job started*)
		ScheduledDowntimeRate : REAL; (*Percentage of scheduled downtime [%] since this job started*)
		UnscheduledDowntimeRate : REAL; (*Percentage of unscheduled downtime [%] since this job started*)
		NominalProductionTimeRate : REAL; (*Percentage of nominal speed running time[%] since this job started*)
		TargetPieces : UDINT; (*Specifies the target quantity of products to be produced by the machine at nominal speed*)
		TotalPieces : UDINT; (*Counter for total products since this job started*)
		GoodPieces : UDINT; (*Counter for good products since this job started*)
		RejectPieces : UDINT; (*Counter for reject products since this job started*)
		BadPieceRate : REAL; (*Percentage of bad products [%] since this job started*)
		CurrentProductionRate : REAL; (*Production rate since this job started [products / h]*)
		CurrentUser : STRING[50]; (*Currently active user*)
		AdditionalData : STRING[EVENT_ADDITONAL_DATA_LEN]; (*Additional data information*)
	END_STRUCT;
	exCoreInternalRecordEnum :
		(
		RecordTypeJob := 0,
		RecordTypeShift := 1,
		RecordTypeNoShift := 2,
		RecordTypeUptime := 3,
		RecordTypeDowntimeScheduled := 4,
		RecordTypeDowntimeUnscheduled := 5,
		RecordTypeUserChange := 6,
		RecordTypeTimeline := 10
		);
	exCoreInternalExportEnum :
		(
		ExportTypeJob,
		ExportTypeShift,
		ExportTypeTimeline
		);
	exConfigInternalDataType : 	STRUCT
		State : exAssetIntStateEnum;
		StateError : exAssetIntStateEnum := exASSETINT_STATE_NONE;
		ReadConfiguration : ReadConfiguration;
		WriteConfiguration : WriteConfiguration;
	END_STRUCT;
	exUIInternalDataType : 	STRUCT
		RecordStart : DINT; (*Visible list is starting from this index*)
		RecordCount : UINT; (*Total number of items*)
		RecordCountOld : UINT; (*Old record number is required for DESC list*)
		RecordData : exCoreInternalRecordType;
		TimeSeconds : UDINT;
		TimeLongest : UDINT;
		SortingStartTimeOld : exAssetIntUISortingEnum := exASSETINT_SORTING_ASC;
		DT_TO_DTStructure_0 : DTStructure;
		x : UDINT;
		y : UDINT;
		State : exAssetIntStateEnum;
		StateError : exAssetIntStateEnum := exASSETINT_STATE_NONE;
	END_STRUCT;
	exAssetIntLinkType : 	STRUCT
		Version : USINT; (*Data structure version*)
		MemoryDb : UDINT; (*Database memory*)
		MemoryJob : UDINT; (*Job data memory*)
		MemoryShift : UDINT; (*Shift data memory*)
		MemoryTimeline : UDINT; (*Timeline data memory*)
		StatsLastCall : DTStructure; (*Date and time when the stats were last calculated*)
		Configuration : exAssetIntCoreConfigType; (*Configuration structure*)
		RecordCount : UINT; (*Number of total records*)
		IsCoreActive : BOOL; (*Core function block is ready*)
		RefreshJobUI : BOOL; (*Update job stats in UI*)
		RefreshShiftUI : BOOL; (*Update shift stats in UI*)
		RefreshTimelineUI : BOOL; (*Update timeline stats in UI*)
		ShiftStatistics : exAssetIntShiftStatisticsType; (*Current shift stats*)
		ShiftTotalTime : LREAL; (*Milliseconds the job is running*)
		ShiftDowntimeScheduled : UDINT; (*Milliseconds of scheduled downtime*)
		ShiftDowntimeUnscheduled : UDINT; (*Milliseconds of unscheduled downtime*)
		ShiftSecondsToEnd : UDINT;
		JobStatistics : exAssetIntJobStatisticsType; (*Current job stats*)
		JobTotalTime : LREAL; (*Milliseconds the job is running*)
		JobDowntimeScheduled : UDINT; (*Milliseconds of scheduled downtime*)
		JobDowntimeUnscheduled : UDINT; (*Milliseconds of unscheduled downtime*)
		ShiftId : SINT := -1; (*Index of shift configuration*)
		ProductionStateStart : DATE_AND_TIME; (*Current state beginning*)
		ProductionState : exAssetIntUIProductionStateEnum; (*Current state*)
		ProductionTotalTime : LREAL; (*Milliseconds the state is running*)
		ProductionUserName : STRING[50]; (*Currently active user*)
		ProductionShiftName : STRING[20]; (*ShiftName for this timeline*)
		ProductionJobName : STRING[20]; (*Job name for this timeline*)
		ProductionDowntime : exAssetIntDowntimeEnum; (*Downtime for this timeline*)
		ProductionDowntimeReason : STRING[50]; (*Donwtime reason for this timeline*)
	END_STRUCT;
END_TYPE

(*Enum type*)

TYPE
	exAssetIntStateEnum :
		(
		exASSETINT_STATE_INIT_1 := 1, (*Init state*)
		exASSETINT_STATE_INIT_2 := 2, (*Init state*)
		exASSETINT_STATE_INIT_3 := 3, (*Init state*)
		exASSETINT_STATE_INIT_4 := 4, (*Init state*)
		exASSETINT_STATE_INIT_5 := 5, (*Init state*)
		exASSETINT_STATE_IDLE := 10, (*Wait for command and collect data*)
		exASSETINT_STATE_STORE_EVENT := 20, (*Store new event data*)
		exASSETINT_STATE_EXPORT_EVENTS := 21, (*Export all events*)
		exASSETINT_STATE_UI_BUFFER := 30, (*Copy job data from global buffer to UI buffer*)
		exASSETINT_STATE_UI_DATA := 31, (*Generate UI data*)
		exASSETINT_STATE_SAVE_CFG := 40, (*Save configuration*)
		exASSETINT_STATE_LOAD_CFG := 41, (*Load configuration*)
		exASSETINT_STATE_SAVE_LINK := 50, (*Save internal data*)
		exASSETINT_STATE_LOAD_LINK := 51, (*Load internal data*)
		exASSETINT_STATE_ERROR := 90, (*Error state*)
		exASSETINT_STATE_NONE := 99 (*Empty state*)
		);
	exAssetIntLogLevelEnum :
		(
		exASSETINT_LOG_OFF := 0, (*Logging is disabled*)
		exASSETINT_LOG_ERROR := 1, (*Only log errors*)
		exASSETINT_LOG_INFO := 2, (*Also log information*)
		exASSETINT_LOG_ALL := 3 (*Log everything*)
		);
	exAssetIntBufferOffsets :
		(
		exASSETINT_BUFFER_MEMORY := 0
		);
	exAssetIntUIStatusEnum :
		(
		exASSETINT_UI_STATUS_IDLE := 0, (*Status: Idle, Waiting for command*)
		exASSETINT_UI_STATUS_UPDATE := 1, (*Status: Updating UIConnect structer*)
		exASSETINT_UI_STATUS_FILTER := 2 (*Status: Showing filter-dialog*)
		);
	exAssetIntMemoryEnum :
		(
		exASSETINT_MEM_DB := 0, (*Database memory*)
		exASSETINT_MEM_JOB := 1, (*Job working memory*)
		exASSETINT_MEM_SHIFT := 2, (*Shift working memory*)
		exASSETINT_MEM_TIMELINE := 3 (*Timeline working memory*)
		);
	exAssetIntDowntimeEnum :
		(
		exASSETINT_NO_DOWNTIME := 0, (*No downtime active = uptime*)
		exASSETINT_SCHEDULED_DOWNTIME := 1, (*Additional scheduled downtime (e.g. monthly maintenance)*)
		exASSETINT_UNSCHEDULED_DOWNTIME := 2 (*Unscheduled downtime (e.g. machine fault)*)
		);
	exComSeveritiesEnum :
		(
		exCOM_SEV_SUCCESS := 0, (*Success - no error*)
		exCOM_SEV_INFORMATIONAL := 1, (*Severity: Informational*)
		exCOM_SEV_WARNING := 2, (*Severity: Warning*)
		exCOM_SEV_ERROR := 3 (*Severity: Error*)
		);
END_TYPE

(*Config type*)

TYPE
	exAssetIntCoreConfigType : 	STRUCT
		CalculationTimeBase : UDINT := 1000; (*Cycle time for calculating the current production rate*)
		Shifts : ARRAY[0..4]OF exAssetIntShiftParType := [5(0)]; (*Shift schedule in detailed*)
		Export : exAssetIntExportType; (*Configuration for export*)
	END_STRUCT;
	exAssetIntExportType : 	STRUCT
		JobStatistics : BOOL := TRUE; (*Export the job statistics or not.*)
		JobStatisticsFileNamePattern : STRING[50] := 'JobStatistics_%Y_%m_%d_%H_%M.csv'; (*Pattern for export job statistics file.*)
		ShiftStatistics : BOOL := TRUE; (*Export the shift statistics or not.*)
		ShiftStatisticsFileNamePattern : STRING[50] := 'ShiftStatistics_%Y_%m_%d_%H_%M.csv'; (*Pattern for export shift statistics file.*)
		Timeline : BOOL := TRUE; (*Export the timeline statistics or not.*)
		TimelineFileNamePattern : STRING[50] := 'Timeline_%Y_%m_%d_%H_%M.csv'; (*Pattern for export timeline  file.*)
		TimestampPattern : STRING[50] := '%Y-%m-%d %H:%M:%S'; (*Timestamp pattern in exported file.*)
		DecimalDigits : UINT := 2; (*Specifies how many decimal positions are saved*)
		ColumnSeparator : STRING[1] := ','; (*Delimiter used to split up PVs in the .csv file*)
		DecimalMark : STRING[1] := '.'; (*Character to be used for the decimal separator*)
	END_STRUCT;
	exAssetIntShiftParType : 	STRUCT
		Name : STRING[20]; (*Shift name*)
		TotalTime : exAssetIntTimeSlotType; (*Total time of one shift*)
		ScheduledDowntime : ARRAY[0..9]OF exAssetIntScheduledDowntimeType; (*Scheduled downtime in one shift*)
	END_STRUCT;
	exAssetIntTimeSlotType : 	STRUCT
		Start : TIME_OF_DAY; (*Start time.*)
		End : TIME_OF_DAY; (*End time*)
	END_STRUCT;
	exAssetIntScheduledDowntimeType : 	STRUCT
		Reason : STRING[50]; (*Downtime reason*)
		Start : TIME_OF_DAY; (*Start time.*)
		End : TIME_OF_DAY; (*End time*)
	END_STRUCT;
END_TYPE

(*Parameter type*)

TYPE
	exAssetIntParType : 	STRUCT
		NominalProductionRate : REAL := 0.0; (*Nominal production rate [products / h]*)
		Job : STRING[20] := 'Job1'; (*Currently active production job*)
		CurrentUser : STRING[50]; (*Currently logged in user*)
		AdditionalData : STRING[255]; (*Additional data to be logged*)
	END_STRUCT;
END_TYPE

(*UI type*)

TYPE
	exAssetIntUITrendType : 	STRUCT
		SaexleData : ARRAY[0..365]OF REAL; (*FB->VC:Saexle data for trend data*)
		SaexleRate : UDINT; (*FB->VC:Saexle rate datapoint for trend data*)
		SaexleCount : UDINT; (*FB->VC:Saexle count datapoint for trend data*)
		SaexleDateTime : DATE_AND_TIME; (*FB->VC:Saexle DataTime datapoint for trend data*)
		MinValue : REAL; (*FB->VC:Min.value datapoint for trend data*)
		MaxValue : REAL; (*FB->VC:Max.value datapoint for trend data*)
		HideCurve : INT; (*FB->VC:Hide the curve if set to 1, status datapoint for trend curve*)
		TimeZoom : REAL; (*FB->VC:Zoom datapoint for trend time scale.*)
		TimeScroll : REAL; (*FB->VC:Scoll datapoint for trend time scale.*)
	END_STRUCT;
	exAssetIntUIShiftListType : 	STRUCT
		ShiftNames : ARRAY[0..5]OF STRING[20]; (*FB->VC: Shift names, *)
		SelectedIndex : UINT; (*VC->FB: Selection index for ShiftList.*)
		MaxSelection : USINT;
	END_STRUCT;
	exAssetIntTrendUIConnectType : 	STRUCT
		Status : exAssetIntUIStatusEnum; (*Status of UI function block*)
		ScheduledDowntimeRate : exAssetIntUITrendType; (*Trend for scheduled downtime rate*)
		UnscheduledDowntimeRate : exAssetIntUITrendType; (*Trend for unscheduled downtime rate*)
		NominalProductionRate : exAssetIntUITrendType; (*Trend for nominal production rate*)
		BadPieceRate : exAssetIntUITrendType; (*Trend for bad piece rate*)
		ShiftList : exAssetIntUIShiftListType; (*Determine which shift in the day is shown in the trend*)
		Filter : exAssetIntUIFilterType; (*Output filter.*)
	END_STRUCT;
	exAssetIntUITimelineOutputType : 	STRUCT
		StartTime : ARRAY[0..UI_TIMELINE_IDX]OF DATE_AND_TIME; (*FB->VC:Start time of this state*)
		ShiftName : ARRAY[0..UI_TIMELINE_IDX]OF STRING[20]; (*FB->VC:Shift name*)
		JobName : ARRAY[0..UI_TIMELINE_IDX]OF STRING[20]; (*FB->VC:Job name*)
		ProductionState : ARRAY[0..UI_TIMELINE_IDX]OF exAssetIntUIProductionStateEnum; (*FB->VC:Production state*)
		Reason : ARRAY[0..UI_TIMELINE_IDX]OF STRING[50]; (*FB->VC:Reason of this state*)
		Duration : ARRAY[0..UI_TIMELINE_IDX]OF exAssetIntTimeType; (*FB->VC:Duration of this state*)
		DurationBar : ARRAY[0..UI_TIMELINE_IDX]OF exAssetIntUITimeBargraphType; (*FB->VC:Duration of this state in a graphic way*)
		RangeStart : REAL; (*Displayed range: Start %*)
		RangeEnd : REAL; (*Displayed range: End %*)
		PageUp : BOOL; (*Command: Page Up (Scroll Up)*)
		StepUp : BOOL; (*Command: Line Up (Scroll Up)*)
		StepDown : BOOL; (*Command: Line Down (Scroll Down)*)
		PageDown : BOOL; (*Command: Page Down (Scroll Down)*)
	END_STRUCT;
	exAssetIntUITimeBargraphType : 	STRUCT
		Duration : UDINT; (*FB->VC:EndValue(lenth) of the scale*)
		Color : UDINT; (*FB->VC:ColorDatapoint of the scale*)
	END_STRUCT;
	exAssetIntTimelineUIConnectType : 	STRUCT
		Status : exAssetIntUIStatusEnum; (*Status of UI function block*)
		Output : exAssetIntUITimelineOutputType; (*Output information.*)
		Filter : exAssetIntUIFilterType; (*Output filter.*)
	END_STRUCT;
	exAssetIntTimeType : 	STRUCT
		Hours : UDINT; (*Numbers of hours*)
		Minutes : USINT; (*Numbers of minutes within an hour*)
		Seconds : USINT; (*Numbers of seconds within a minute*)
	END_STRUCT;
	exAssetIntShiftListUIConnectType : 	STRUCT
		Status : exAssetIntUIStatusEnum; (*Status of UI function block*)
		Output : exAssetIntUIShiftListOutputType; (*Output information.*)
		Filter : exAssetIntUIFilterType; (*Output filter.*)
	END_STRUCT;
	exAssetIntUIShiftListOutputType : 	STRUCT
		StartTime : ARRAY[0..UI_SHIFT_LIST_IDX]OF DATE_AND_TIME; (*Start time list*)
		EndTime : ARRAY[0..UI_SHIFT_LIST_IDX]OF DATE_AND_TIME; (*End time list*)
		ShiftName : ARRAY[0..UI_SHIFT_LIST_IDX]OF STRING[20]; (*Shift ID list*)
		CurrentUser : ARRAY[0..UI_SHIFT_LIST_IDX]OF STRING[50]; (*Currently active user*)
		AdditionalData : ARRAY[0..UI_SHIFT_LIST_IDX]OF STRING[255]; (*Additional data information*)
		TargetPieces : ARRAY[0..UI_SHIFT_LIST_IDX]OF UDINT; (*Target pieces list*)
		TotalPieces : ARRAY[0..UI_SHIFT_LIST_IDX]OF UDINT; (*Total pieces list*)
		GoodPieces : ARRAY[0..UI_SHIFT_LIST_IDX]OF UDINT; (*Good pieces list*)
		RejectPieces : ARRAY[0..UI_SHIFT_LIST_IDX]OF UDINT; (*Reject pieces list*)
		BadPieceRate : ARRAY[0..UI_SHIFT_LIST_IDX]OF REAL; (*bad piece rate list*)
		TotalTime : ARRAY[0..UI_SHIFT_LIST_IDX]OF exAssetIntTimeType; (*Total time list*)
		ScheduledDowntime : ARRAY[0..UI_SHIFT_LIST_IDX]OF exAssetIntTimeType; (*Scheduled Downtime list*)
		UnscheduledDowntime : ARRAY[0..UI_SHIFT_LIST_IDX]OF exAssetIntTimeType; (*Unscheduled Downtime list*)
		Uptime : ARRAY[0..UI_SHIFT_LIST_IDX]OF exAssetIntTimeType; (*Uptime list*)
		GoodProductionTime : ARRAY[0..UI_SHIFT_LIST_IDX]OF exAssetIntTimeType; (*Good production time list*)
		NominalProductionTime : ARRAY[0..UI_SHIFT_LIST_IDX]OF exAssetIntTimeType; (*nominal production time list*)
		NominalProductionRate : ARRAY[0..UI_SHIFT_LIST_IDX]OF REAL; (*nominal production rate list*)
		ShiftProductionRate : ARRAY[0..UI_SHIFT_LIST_IDX]OF REAL; (*Shift production rate list*)
		ScheduledDowntimeRate : ARRAY[0..UI_SHIFT_LIST_IDX]OF REAL; (*scheduled downtime rate list*)
		UnscheduledDowntimeRate : ARRAY[0..UI_SHIFT_LIST_IDX]OF REAL; (*unscheduled downtime rate list*)
		ProductionRate : ARRAY[0..UI_SHIFT_LIST_IDX]OF REAL; (*current production rate list*)
		RangeStart : REAL; (*Displayed range: Start %*)
		RangeEnd : REAL; (*Displayed range: End %*)
		PageUp : BOOL; (*Command: Page Up (Scroll Up)*)
		StepUp : BOOL; (*Command: Line Up (Scroll Up)*)
		StepDown : BOOL; (*Command: Line Down (Scroll Down)*)
		PageDown : BOOL; (*Command: Page Down (Scroll Down)*)
		IdealProductionRate : ARRAY[0..UI_SHIFT_LIST_IDX]OF REAL; (*ideal production rate list*)
		JobName : ARRAY[0..UI_SHIFT_LIST_IDX]OF STRING[20]; (*Job name list*)
	END_STRUCT;
	exAssetIntUIShiftListJobType : 	STRUCT  (*Jobs within one shift*)
		Name : ARRAY[0..9]OF STRING[20]; (*Name of the job*)
	END_STRUCT;
	exAssetIntListUISetupType : 	STRUCT
		ScrollWindow : USINT := 0; (*Scroll Window (overlap for PageUp/Down)*)
		SortingStartTime : exAssetIntUISortingEnum := exASSETINT_SORTING_DESC;
	END_STRUCT;
	exAssetIntJobListUIConnectType : 	STRUCT
		Status : exAssetIntUIStatusEnum; (*Status of UI function block*)
		Output : exAssetIntUIJobListOutputType; (*Output information.*)
		Filter : exAssetIntUIFilterType; (*Output filter.*)
	END_STRUCT;
	exAssetIntUIJobListOutputType : 	STRUCT
		JobStartTime : ARRAY[0..UI_JOB_LIST_IDX]OF DATE_AND_TIME; (*Job start time list*)
		JobEndTime : ARRAY[0..UI_JOB_LIST_IDX]OF DATE_AND_TIME; (*Job end time list*)
		JobName : ARRAY[0..UI_JOB_LIST_IDX]OF STRING[20]; (*Job name list*)
		CurrentUser : ARRAY[0..UI_JOB_LIST_IDX]OF STRING[50]; (*Currently active user*)
		AdditionalData : ARRAY[0..UI_JOB_LIST_IDX]OF STRING[255]; (*Additional data information*)
		TotalPieces : ARRAY[0..UI_JOB_LIST_IDX]OF UDINT; (*Total pieces list*)
		GoodPieces : ARRAY[0..UI_JOB_LIST_IDX]OF UDINT; (*Good pieces list*)
		RejectPieces : ARRAY[0..UI_JOB_LIST_IDX]OF UDINT; (*Reject pieces list*)
		BadPieceRate : ARRAY[0..UI_JOB_LIST_IDX]OF REAL; (*bad piece rate list*)
		TotalTime : ARRAY[0..UI_JOB_LIST_IDX]OF exAssetIntTimeType; (*Total time list*)
		ScheduledDowntime : ARRAY[0..UI_JOB_LIST_IDX]OF exAssetIntTimeType; (*Scheduled Downtime list*)
		UnscheduledDowntime : ARRAY[0..UI_JOB_LIST_IDX]OF exAssetIntTimeType; (*Unscheduled Downtime list*)
		Uptime : ARRAY[0..UI_JOB_LIST_IDX]OF exAssetIntTimeType; (*Uptime list*)
		GoodProductionTime : ARRAY[0..UI_JOB_LIST_IDX]OF exAssetIntTimeType; (*Good production time list*)
		NominalProductionTime : ARRAY[0..UI_JOB_LIST_IDX]OF exAssetIntTimeType; (*nominal production time list*)
		NominalProductionRate : ARRAY[0..UI_JOB_LIST_IDX]OF REAL; (*nominal production rate list*)
		ScheduledDowntimeRate : ARRAY[0..UI_JOB_LIST_IDX]OF REAL; (*scheduled downtime rate list*)
		UnscheduledDowntimeRate : ARRAY[0..UI_JOB_LIST_IDX]OF REAL; (*unscheduled downtime rate list*)
		ProductionRate : ARRAY[0..UI_JOB_LIST_IDX]OF REAL; (*current production rate list*)
		RangeStart : REAL; (*Displayed range: Start %*)
		RangeEnd : REAL; (*Displayed range: End %*)
		PageUp : BOOL; (*Command: Page Up (Scroll Up)*)
		StepUp : BOOL; (*Command: Line Up (Scroll Up)*)
		StepDown : BOOL; (*Command: Line Down (Scroll Down)*)
		PageDown : BOOL; (*Command: Page Down (Scroll Down)*)
		ShiftName : ARRAY[0..UI_JOB_LIST_IDX]OF STRING[20]; (*Shift ID list*)
	END_STRUCT;
	exAssetIntUISortingEnum :
		(
		exASSETINT_SORTING_ASC := 0, (*Sorting ascending*)
		exASSETINT_SORTING_DESC := 1 (*Sorting descending*)
		);
	exAssetIntUIProductionStateEnum :
		(
		exASSETINT_STATE_NO_SHIFT_ACTIVE := 0, (*Inactive state*)
		exASSETINT_STATE_UPTIME := 1, (*Uptime state*)
		exASSETINT_STATE_SCHDL_DOWNTIME := 2, (*Scheduled downtime state*)
		exASSETINT_STATE_UNSCH_DOWNTIME := 3 (*Unscheduled downtime state*)
		);
	exAssetIntUICurrDTFilterType : 	STRUCT
		Enable : BOOL; (*Enable Filter*)
		DateTime : DATE_AND_TIME; (*Date and time of filter*)
	END_STRUCT;
	exAssetIntUISetDTFilterType : 	STRUCT
		Enable : BOOL; (*Enable Filter*)
		Year : UINT; (*Date&Time: Year*)
		Month : USINT; (*Date&Time: Month*)
		Day : USINT; (*Date&Time: Day*)
		Hour : USINT; (*Date&Time: Hour*)
		Minute : USINT; (*Date&Time: Minute*)
	END_STRUCT;
	exAssetIntUIFilterDialogType : 	STRUCT
		LayerStatus : UINT := UI_LAYER_HIDE; (*			Filter.Dialog.LayerStatus := UI_LAYER_HIDE;
*)
		From : exAssetIntUISetDTFilterType; (*Display entries from given date&time*)
		Until : exAssetIntUISetDTFilterType; (*Display entries until given date&time*)
		Confirm : BOOL;
		Cancel : BOOL;
	END_STRUCT;
	exAssetIntUIFilterType : 	STRUCT
		ShowDialog : BOOL;
		Dialog : exAssetIntUIFilterDialogType; (*Dialog-data to change filter-settings*)
		Current : exAssetIntUICurrentFilterType; (*Currently active filter settings*)
		DefaultLayerStatus : UINT;
	END_STRUCT;
	exAssetIntUICurrentFilterType : 	STRUCT
		From : exAssetIntUICurrDTFilterType; (*Starting time of current filter*)
		Until : exAssetIntUICurrDTFilterType; (*End time of current filter*)
	END_STRUCT;
END_TYPE

(*Info type*)

TYPE
	exAssetIntJobStatisticsType : 	STRUCT
		JobName : STRING[20]; (*Job name.*)
		StartTime : DATE_AND_TIME;
		TotalTime : exAssetIntTimeType; (*Total time since this job started*)
		ScheduledDowntime : exAssetIntTimeType; (*Scheduled downtime since this job started*)
		UnscheduledDowntime : exAssetIntTimeType; (*Unsheduled downtime since this job started*)
		Uptime : exAssetIntTimeType; (*Uptime since this job started*)
		NominalProductionTime : exAssetIntTimeType; (*Time of production at nominal speed since this job started*)
		GoodProductionTime : exAssetIntTimeType; (*Time of good production since this job started*)
		ScheduledDowntimeRate : REAL; (*Percentage of scheduled downtime [%] since this job started*)
		UnscheduledDowntimeRate : REAL; (*Percentage of unscheduled downtime [%] since this job started*)
		NominalProductionTimeRate : REAL; (*Percentage of nominal speed running time[%] since this job started*)
		TotalPieces : UDINT; (*Counter for total products since this job started*)
		GoodPieces : UDINT; (*Counter for good products since this job started*)
		RejectPieces : UDINT; (*Counter for reject products since this job started*)
		BadPieceRate : REAL; (*Percentage of bad products [%] since this job started*)
		CurrentProductionRate : REAL; (*Production rate since this job started [products / h]*)
		CurrentUser : STRING[50]; (*Currently active user*)
		AdditionalData : STRING[EVENT_ADDITONAL_DATA_LEN]; (*Additional data information*)
	END_STRUCT;
	exAssetIntShiftStatisticsType : 	STRUCT
		ShiftName : STRING[20]; (*Shift name.*)
		StartTime : DATE_AND_TIME;
		TotalTime : exAssetIntTimeType; (*Total time since this shift started*)
		ScheduledDowntime : exAssetIntTimeType; (*Scheduled downtime since this shift started*)
		UnscheduledDowntime : exAssetIntTimeType; (*Unsheduled downtime since this shift started*)
		Uptime : exAssetIntTimeType; (*Uptime since this shift started*)
		GoodProductionTime : exAssetIntTimeType; (*Time of good production since this shift started*)
		NominalProductionTime : exAssetIntTimeType; (*Time of production at nominal speed since this shift started*)
		ScheduledDowntimeRate : REAL; (*Percentage of scheduled downtime [%] since this shift started*)
		UnscheduledDowntimeRate : REAL; (*Percentage of unscheduled downtime [%] since this shift started*)
		NominalProductionTimeRate : REAL; (*Percentage of nominal speed running time[%] since this shift started*)
		TargetPieces : UDINT; (*Counter for target products since this shift started*)
		TotalPieces : UDINT; (*Counter for total products since this shift started*)
		GoodPieces : UDINT; (*Counter for good products since this shift started*)
		RejectPieces : UDINT; (*Counter for reject products since this shift started*)
		BadPieceRate : REAL; (*Percentage of bad products [%] since this shift started*)
		CurrentProductionRate : REAL; (*Production rate since this shift started [products / h]*)
		CurrentUser : STRING[50]; (*Currently active user*)
		AdditionalData : STRING[255]; (*Additional data information*)
		IdealProductionRate : REAL; (*Ideal production rate*)
	END_STRUCT;
	exAssetIntCoreInfoType : 	STRUCT
		ShiftStatistics : exAssetIntShiftStatisticsType; (*Shift statistics*)
		JobStatistics : exAssetIntJobStatisticsType; (*Job statistics*)
		Diag : exAssetIntDiagType; (*Additional diagnostic information*)
	END_STRUCT;
	exAssetIntInfoType : 	STRUCT
		Diag : exAssetIntDiagType; (*Additional diagnostic information*)
	END_STRUCT;
	exAssetIntDiagType : 	STRUCT
		StatusID : exAssetIntStatusIDType; (*Segmented StatusID output*)
	END_STRUCT;
	exAssetIntStatusIDType : 	STRUCT
		ID : exAssetIntErrorEnum; (*StatusID as enumerator*)
		Severity : exComSeveritiesEnum; (*Severity of the error*)
		Code : UINT; (*Error code*)
	END_STRUCT;
END_TYPE
```

#### Constants.var - Exported constants
```iecst
(*------------------------------------------------------------------------------------------------------------------------------------------------------------------------------------------------------------------------------------------------------------------------------------------------------------------------------------------------------*)
(*General constants*)
(*------------------------------------------------------------------------------------------------------------------------------------------------------------------------------------------------------------------------------------------------------------------------------------------------------------------------------------------------------*)
VAR CONSTANT
	CORE_EVENT_NUM_MAX : UINT := 500; (*Maximum number of events*)
	CORE_EVENT_DIR_MAX : UINT := 1000; (*Maximum number of events in one directory*)
	EVENT_ADDITONAL_DATA_LEN : UINT := 100; (*Length of the event comment*)
END_VAR
(*------------------------------------------------------------------------------------------------------------------------------------------------------------------------------------------------------------------------------------------------------------------------------------------------------------------------------------------------------*)
(*Export constants*)
(*------------------------------------------------------------------------------------------------------------------------------------------------------------------------------------------------------------------------------------------------------------------------------------------------------------------------------------------------------*)
VAR CONSTANT
	EXPORT_BUFFER : UINT := 500; (*Length of the buffer for the event export*)
	EXPORT_JOB_TITEL : STRING[100] := 'AssetInt Job Statistics Export File'; (*Export file header*)
	EXPORT_SHIFT_TITEL : STRING[100] := 'AssetInt Shift Statistics Export File'; (*Export file header*)
	EXPORT_TIMELINE_TITEL : STRING[100] := 'AssetInt Timeline Statistics Export File'; (*Export file header*)
	EXPORT_JOB_HEADER : STRING[400] := 'Job Start Time;Job End Time;Job Name;Current User;Additional Data;Total Pieces;Good Pieces;Reject Pieces;Bad Piece Rate;Total Time;Scheduled Downtime;Unscheduled Downtime;Uptime;Good Production Time;Nominal Production Time;Nominal Production Time Rate;Scheduled Downtime Rate;Unscheduled Downtime Rate;Production Rate;Shift Name'; (*Export file column headers*)
	EXPORT_SHIFT_HEADER : STRING[400] := 'Job Start Time;Job End Time;Job Name;Current User;Additional Data;Total Pieces;Good Pieces;Reject Pieces;Bad Piece Rate;Total Time;Scheduled Downtime;Unscheduled Downtime;Uptime;Good Production Time;Nominal Production Time;Nominal Production Time Rate;Scheduled Downtime Rate;Unscheduled Downtime Rate;Production Rate;Shift Name'; (*Export file column headers*)
	EXPORT_TIMELINE_HEADER : STRING[400] := 'Start Time;Shift ID;Production State;Reason;Duration;Job Name'; (*Export file column headers*)
END_VAR
(*------------------------------------------------------------------------------------------------------------------------------------------------------------------------------------------------------------------------------------------------------------------------------------------------------------------------------------------------------*)
(*UI constants*)
(*------------------------------------------------------------------------------------------------------------------------------------------------------------------------------------------------------------------------------------------------------------------------------------------------------------------------------------------------------*)
VAR CONSTANT
	UI_SHIFT_LIST_IDX : UINT := 8; (*Max index for list box entries for shift data*)
	UI_TIMELINE_IDX : UINT := 8; (*Max index for list box entries for timeline data*)
	UI_JOB_LIST_IDX : UINT := 8; (*Max index for list box entries for job data*)
	UI_SHIFT_SHOW_JOBS : BOOL := TRUE; (*Show job changes in shift list*)
END_VAR
(*------------------------------------------------------------------------------------------------------------------------------------------------------------------------------------------------------------------------------------------------------------------------------------------------------------------------------------------------------*)
(*Logger constants*)
(*------------------------------------------------------------------------------------------------------------------------------------------------------------------------------------------------------------------------------------------------------------------------------------------------------------------------------------------------------*)
VAR CONSTANT
	LOG_LEN : UINT := 100; (*Length of one log entry (minimum size is 50)*)
	LOG_NUM : UINT := 50; (*Number of log entries*)
	LOG_LEVEL : exAssetIntLogLevelEnum := exASSETINT_LOG_ALL; (*Define log level details*)
	CHAR_RETURN : USINT := 13; (*Carriage return*)
END_VAR
(*------------------------------------------------------------------------------------------------------------------------------------------------------------------------------------------------------------------------------------------------------------------------------------------------------------------------------------------------------*)
(*Error codes*)
(*------------------------------------------------------------------------------------------------------------------------------------------------------------------------------------------------------------------------------------------------------------------------------------------------------------------------------------------------------*)
VAR CONSTANT
	ERR_ASSET_LINK : DINT := -1064239102; (*Input exLink is 0 pointer*)
	ERR_ASSET_TEMP_MEMORY : DINT := -1064136704; (*No temporary memory available, make sure core function block is enabled*)
	ERR_ASSET_INF_WAIT_CORE_FB : DINT := 1083346949; (*This component can only become active if MpAssetIntCore is active.*)
	ERR_ASSET_READ_RECORD_SIZE : DINT := -2138009590; (*Record size is not correct during reading event data*)
	ERR_ASSET_READ_CRC : DINT := 100000; (*Record CRC error during reading event data*)
	ERR_ASSET_CONFIG : DINT := -1064239096; (*Configuration link is 0 pointer*)
	ERR_ASSET_SHIFT_CALC : DINT := -1064239097; (*Invalid shift configured*)
END_VAR
```

#### exAssetInt.fun - Exported functions and function blocks
```iecst
FUNCTION_BLOCK exAssetIntCore (*mapp function block which can be used for asset intensity calculation.*) (* $GROUP=mapp Services,$CAT=Asset Intensity,$GROUPICON=Icon_mapp.png,$CATICON=Icon_exOee.png *)
	VAR_INPUT
		exLink : REFERENCE TO exAssetIntLinkType; (*Incoming communication handle (mapp standard interface)*) (* *) (*#PAR#;*)
		Enable : BOOL; (*Enables/Disables the function block (mapp standard interface)*) (* *) (*#PAR#;*)
		ErrorReset : BOOL; (*Resets all function block errors (mapp standard interface)*) (* *) (*#PAR#;*)
		Parameters : REFERENCE TO exAssetIntParType; (*Function block parameters (mapp standard interface)*) (* *) (*#PAR#; *)
		Logger : UDINT;
		Configuration : REFERENCE TO exAssetIntCoreConfigType;
		Update : BOOL; (*Updates the parameters (mapp standard interface)*) (* *) (*#PAR#; *)
		Downtime : exAssetIntDowntimeEnum; (*The machine is in down time*) (* *) (*#CMD#; *)
		DowntimeReason : REFERENCE TO STRING[50]; (*The reason for down time*) (* *) (*#CMD#; *)
		PieceCounter : UDINT; (*Total pieces counter.*) (* *) (*#CMD#; *)
		RejectCounter : UDINT; (*Reject pieces counter*) (* *) (*#CMD#; *)
		DeviceName : REFERENCE TO STRING[50]; (*Address of the exported device name*) (* *) (*#CMD#; *)
		StorageName : REFERENCE TO STRING[50]; (*Address of the storage device name*) (* *) (*#CMD#; *)
		Export : BOOL; (*Export the saved information to file*) (* *) (*#CMD#; *)
		Reset : BOOL; (*Reset the data buffer*) (* *) (*#CMD#; *)
	END_VAR
	VAR_OUTPUT
		Active : BOOL; (*Function block is active (mapp standard interface)*) (* *) (*#PAR#;*)
		Error : BOOL; (*Indicates an error (mapp standard interface)*) (* *) (*#PAR#;*)
		StatusID : DINT; (*Error/Status information (mapp standard interface)*) (* *) (*#PAR#; *)
		UpdateDone : BOOL; (*Update of parameters done (mapp standard interface)*) (* *) (*#PAR#; *)
		CommandBusy : BOOL; (*Function block is busy processing a command*) (* *) (*#CMD#OPT#;*)
		CommandDone : BOOL; (*True if a command finshed successfully.*) (* *) (*#CMD#OPT#;*)
		CurrentProductionRate : REAL; (*Current production rate [products / h] based on calculation time base*) (* *) (*#CYC#*)
		ScheduledDowntimeRate : REAL; (*Percentage of scheduled downtime [%]*) (* *) (*#CYC#;*)
		UnscheduledDowntimeRate : REAL; (*Percentage of unscheduled downtime [%]*) (* *) (*#CYC#;*)
		NominalProductionTimeRate : REAL; (*Percentage of running time at nominal production speed [%]*) (* *) (*#CYC#;*)
		BadPieceRate : REAL; (*Percentage of bad products [%]*) (* *) (*#CYC#;*)
		ExportDone : BOOL; (*Export command was succesfuly finished*) (* *) (*#CMD#; *)
		Info : exAssetIntCoreInfoType; (*Provide any further useful information as function block output.(mapp standard interface)*) (* *) (*#CMD#; *)
	END_VAR
	VAR
		Internal : {REDUND_UNREPLICABLE} exCoreInternalDataType; (*Internal data*)
		zzEdge00000 : BOOL;
		zzEdge00001 : BOOL;
		zzEdge00002 : BOOL;
		zzEdge00003 : BOOL;
	END_VAR
END_FUNCTION_BLOCK

FUNCTION_BLOCK exAssetIntCoreConfig
	VAR_INPUT
		exLink : REFERENCE TO exAssetIntLinkType; (*Incoming communication handle (mapp standard interface)*) (* *) (*#PAR#;*)
		Enable : BOOL; (*Enables/Disables the function block (mapp standard interface)*) (* *) (*#PAR#;*)
		ErrorReset : BOOL; (*Resets all function block errors (mapp standard interface)*) (* *) (*#PAR#;*)
		DeviceName : REFERENCE TO STRING[30]; (*Address of the exported device name*) (* *) (*#CMD#; *)
		Configuration : REFERENCE TO exAssetIntCoreConfigType;
		Logger : UDINT;
		Load : {REDUND_UNREPLICABLE} BOOL; (* *) (* *) (*#PAR#;*)
		Save : BOOL; (* *) (* *) (*#PAR#;*)
	END_VAR
	VAR_OUTPUT
		Active : BOOL; (*Function block is active (mapp standard interface)*) (* *) (*#PAR#;*)
		Error : BOOL; (*Indicates an error (mapp standard interface)*) (* *) (*#PAR#;*)
		StatusID : DINT; (*Error/Status information (mapp standard interface)*) (* *) (*#PAR#; *)
		CommandBusy : BOOL; (*Function block is busy processing a command*) (* *) (*#CMD#OPT#;*)
		CommandDone : BOOL; (*True if a command finshed successfully.*) (* *) (*#CMD#OPT#;*)
		Info : exAssetIntInfoType; (*Provide any further useful information as function block output.(mapp standard interface)*) (* *) (*#CMD#; *)
	END_VAR
	VAR
		Internal : {REDUND_UNREPLICABLE} exConfigInternalDataType; (*Internal data*)
		zzEdge00000 : BOOL;
		zzEdge00001 : BOOL;
		zzEdge00002 : BOOL;
	END_VAR
END_FUNCTION_BLOCK

FUNCTION_BLOCK exAssetIntJobListUI (*mapp function block which can be used for showing job statistics in a list *)
	VAR_INPUT
		exLink : REFERENCE TO exAssetIntLinkType; (*Incoming communication handle (mapp standard interface)*) (* *) (*#PAR#;*)
		Enable : BOOL; (*Enables/Disables the function block (mapp standard interface)*) (* *) (*#PAR#;*)
		ErrorReset : BOOL; (*Resets all function block errors (mapp standard interface)*) (* *) (*#PAR#;*)
		Logger : UDINT;
		UISetup : exAssetIntListUISetupType; (*Setup UI connection - must be configured before enabling the FB*) (* *) (*#PAR#; *)
		UIConnect : REFERENCE TO exAssetIntJobListUIConnectType; (*Connection structure for VC4 User interface*) (* *) (*#CMD#; *)
	END_VAR
	VAR_OUTPUT
		Active : BOOL; (*Function block is active (mapp standard interface)*) (* *) (*#PAR#;*)
		Error : BOOL; (*Indicates an error (mapp standard interface)*) (* *) (*#PAR#;*)
		StatusID : DINT; (*Error/Status information (mapp standard interface)*) (* *) (*#PAR#; *)
		Info : exAssetIntInfoType; (*Provide any further useful information as function block output.(mapp standard interface)*) (* *) (*#CMD#; *)
	END_VAR
	VAR
		Internal : {REDUND_UNREPLICABLE} exUIInternalDataType; (*Internal data*)
		zzEdge00000 : BOOL;
	END_VAR
END_FUNCTION_BLOCK

FUNCTION_BLOCK exAssetIntShiftListUI (*mapp function block which can be used for showing shift statistics in a list *)
	VAR_INPUT
		exLink : REFERENCE TO exAssetIntLinkType; (*Incoming communication handle (mapp standard interface)*) (* *) (*#PAR#;*)
		Enable : BOOL; (*Enables/Disables the function block (mapp standard interface)*) (* *) (*#PAR#;*)
		ErrorReset : BOOL; (*Resets all function block errors (mapp standard interface)*) (* *) (*#PAR#;*)
		Logger : UDINT;
		UISetup : exAssetIntListUISetupType; (*Setup UI connection - must be configured before enabling the FB*) (* *) (*#PAR#; *)
		UIConnect : REFERENCE TO exAssetIntShiftListUIConnectType; (*Connection structure for VC4 User interface*) (* *) (*#CMD#; *)
	END_VAR
	VAR_OUTPUT
		Active : BOOL; (*Function block is active (mapp standard interface)*) (* *) (*#PAR#;*)
		Error : BOOL; (*Indicates an error (mapp standard interface)*) (* *) (*#PAR#;*)
		StatusID : DINT; (*Error/Status information (mapp standard interface)*) (* *) (*#PAR#; *)
		Info : exAssetIntInfoType; (*Provide any further useful information as function block output.(mapp standard interface)*) (* *) (*#CMD#; *)
	END_VAR
	VAR
		Internal : {REDUND_UNREPLICABLE} exUIInternalDataType; (*Internal data*)
		zzEdge00000 : BOOL;
	END_VAR
END_FUNCTION_BLOCK

FUNCTION_BLOCK exAssetIntTimelineUI (*mapp function block which can be used for showing shift statistics in a list *)
	VAR_INPUT
		exLink : REFERENCE TO exAssetIntLinkType; (*Incoming communication handle (mapp standard interface)*) (* *) (*#PAR#;*)
		Enable : BOOL; (*Enables/Disables the function block (mapp standard interface)*) (* *) (*#PAR#;*)
		ErrorReset : BOOL; (*Resets all function block errors (mapp standard interface)*) (* *) (*#PAR#;*)
		Logger : UDINT;
		UISetup : exAssetIntListUISetupType; (*Setup UI connection - must be configured before enabling the FB*) (* *) (*#PAR#; *)
		UIConnect : REFERENCE TO exAssetIntTimelineUIConnectType; (*Connection structure for VC4 User interface*) (* *) (*#CMD#; *)
	END_VAR
	VAR_OUTPUT
		Active : BOOL; (*Function block is active (mapp standard interface)*) (* *) (*#PAR#;*)
		Error : BOOL; (*Indicates an error (mapp standard interface)*) (* *) (*#PAR#;*)
		StatusID : DINT; (*Error/Status information (mapp standard interface)*) (* *) (*#PAR#; *)
		Info : exAssetIntInfoType; (*Provide any further useful information as function block output.(mapp standard interface)*) (* *) (*#CMD#; *)
	END_VAR
	VAR
		Internal : {REDUND_UNREPLICABLE} exUIInternalDataType; (*Internal data*)
		zzEdge00000 : BOOL;
	END_VAR
END_FUNCTION_BLOCK

FUNCTION_BLOCK CreateDirStructure
	VAR_INPUT
		Enable : BOOL;
		Device : STRING[50];
		Logger : {REDUND_UNREPLICABLE} UDINT; (*Address of log buffer*)
	END_VAR
	VAR_OUTPUT
		Status : DINT;
	END_VAR
	VAR
		DirCreate_0 : DirCreate;
		TmpStr1 : STRING[100];
		TmpStr2 : STRING[100];
		DirCount : USINT;
		State : USINT;
		zzEdge00000 : BOOL;
	END_VAR
END_FUNCTION_BLOCK

FUNCTION_BLOCK CreateMemory
	VAR_INPUT
		Enable : BOOL;
		Size : UDINT;
		Logger : {REDUND_UNREPLICABLE} UDINT; (*Address of log buffer*)
	END_VAR
	VAR_OUTPUT
		MemoryDb : UDINT;
		MemoryJob : UDINT;
		MemoryShift : UDINT;
		MemoryTimeline : UDINT;
		Status : UINT;
	END_VAR
	VAR
		DatObjCreate_0 : DatObjCreate;
		MemoryType : exAssetIntMemoryEnum;
		TmpStr1 : STRING[100];
		TmpStr2 : STRING[100];
		Cnt : USINT;
		State : USINT;
	END_VAR
END_FUNCTION_BLOCK

FUNCTION_BLOCK ReadConfiguration
	VAR_INPUT
		Enable : BOOL;
		Device : REFERENCE TO STRING[50];
		Logger : {REDUND_UNREPLICABLE} UDINT; (*Address of log buffer*)
		Configuration : exAssetIntCoreConfigType;
	END_VAR
	VAR_OUTPUT
		Status : UINT;
	END_VAR
	VAR
		FileOpen_0 : FileOpen;
		FileClose_0 : FileClose;
		FileRead_0 : FileRead;
		State : USINT;
	END_VAR
END_FUNCTION_BLOCK

FUNCTION_BLOCK WriteConfiguration
	VAR_INPUT
		Enable : BOOL;
		Device : REFERENCE TO STRING[50];
		Logger : UDINT; (*Address of log buffer*)
		Configuration : exAssetIntCoreConfigType;
	END_VAR
	VAR_OUTPUT
		Status : UINT;
	END_VAR
	VAR
		FileCreate_0 : FileCreate;
		FileOpen_0 : FileOpen;
		FileClose_0 : FileClose;
		FileWrite_0 : FileWrite;
		Ident : UDINT;
		State : USINT;
	END_VAR
END_FUNCTION_BLOCK

FUNCTION_BLOCK ReadEventData
	VAR_INPUT
		Enable : BOOL;
		Device : STRING[50];
		Logger : {REDUND_UNREPLICABLE} UDINT; (*Address of log buffer*)
		Memory : UDINT;
	END_VAR
	VAR_OUTPUT
		RecordCount : UINT;
		Status : DINT;
	END_VAR
	VAR
		DirOpen_0 : DirOpen;
		DirReadEx_0 : DirReadEx;
		DirClose_0 : DirClose;
		DirName : STRING[100];
		DirCount : USINT;
		FileOpen_0 : FileOpen;
		FileClose_0 : FileClose;
		FileRead_0 : FileRead;
		FileDelete_0 : FileDelete;
		FileName : STRING[100];
		FileInfo_0 : fiDIR_READ_EX_DATA;
		RecordData : exCoreInternalRecordType;
		TimeFirst : DATE_AND_TIME;
		TmpStr1 : STRING[100];
		TmpStr2 : STRING[100];
		Override : {REDUND_UNREPLICABLE} USINT;
		State : USINT;
		CRC : USINT;
		StatusRead : DINT;
		zzEdge00000 : BOOL;
	END_VAR
END_FUNCTION_BLOCK

FUNCTION_BLOCK WriteEventData
	VAR_INPUT
		Enable : BOOL;
		Device : STRING[50];
		Logger : UDINT; (*Address of log buffer*)
		RecordData : UDINT;
		RecordNext : UINT;
	END_VAR
	VAR_OUTPUT
		Status : DINT;
	END_VAR
	VAR
		FileCreate_0 : FileCreate;
		FileOpen_0 : FileOpen;
		FileClose_0 : FileClose;
		FileWrite_0 : FileWrite;
		RecordDataIntern : exCoreInternalRecordType;
		FileName : STRING[100];
		TmpStr1 : STRING[100];
		TmpStr2 : STRING[10];
		Ident : UDINT;
		State : USINT;
		zzEdge00000 : BOOL;
	END_VAR
END_FUNCTION_BLOCK

FUNCTION_BLOCK ExportEventData
	VAR_INPUT
		Enable : BOOL;
		Device : STRING[50];
		Logger : UDINT; (*Address of log buffer*)
		RecordCount : UDINT;
		Memory : UDINT;
		Configuration : exAssetIntExportType;
	END_VAR
	VAR_OUTPUT
		Status : DINT;
	END_VAR
	VAR
		ExportType : exCoreInternalExportEnum;
		FileDelete_0 : FileDelete;
		FileCreate_0 : FileCreate;
		FileClose_0 : FileClose;
		FileWrite_0 : FileWrite;
		RtcGettime : {REDUND_UNREPLICABLE} RTCtime_typ;
		RecordDataIntern : exCoreInternalRecordType;
		DTStructure_0 : DTStructure;
		FileName : STRING[50];
		TmpStr1 : STRING[50];
		TmpStr2 : STRING[50];
		lrealStr : {REDUND_UNREPLICABLE} LREAL;
		Buffer : STRING[EXPORT_BUFFER];
		Offset : UDINT;
		idx : UDINT;
		State : USINT;
	END_VAR
END_FUNCTION_BLOCK

FUNCTION exAssetIntFilterListUI : UDINT
	VAR_INPUT
		Filter : REFERENCE TO exAssetIntUIFilterType;
		Status : REFERENCE TO exAssetIntUIStatusEnum;
		Logger : UDINT;
	END_VAR
	VAR
		DT_TO_DTStructure_0 : DTStructure;
	END_VAR
END_FUNCTION

FUNCTION exAssetIntScrollListUI : BOOL
	VAR_INPUT
		RecordCount : UDINT;
		ListMaxCount : UINT;
		PageUp : REFERENCE TO BOOL; (*Incoming communication handle (mapp standard interface)*) (* *) (*#PAR#;*)
		PageDown : REFERENCE TO BOOL; (*Incoming communication handle (mapp standard interface)*) (* *) (*#PAR#;*)
		StepUp : REFERENCE TO BOOL; (*Incoming communication handle (mapp standard interface)*) (* *) (*#PAR#;*)
		StepDown : REFERENCE TO BOOL; (*Incoming communication handle (mapp standard interface)*) (* *) (*#PAR#;*)
		RecordStart : REFERENCE TO DINT;
		State : REFERENCE TO exAssetIntStateEnum;
	END_VAR
END_FUNCTION

FUNCTION exAssetIntBufferUI : UDINT
	VAR_INPUT
		Memory : UDINT;
		exLink : exAssetIntLinkType; (*Incoming communication handle (mapp standard interface)*) (* *) (*#PAR#;*)
		SortingStartTime : exAssetIntUISortingEnum;
		Filter : exAssetIntUIFilterType;
		EventType : exCoreInternalRecordEnum;
	END_VAR
	VAR
		RecordData : exCoreInternalRecordType;
		RecordCount : UDINT;
		y : UDINT;
	END_VAR
END_FUNCTION

FUNCTION exAssetIntFilterReset : BOOL
	VAR_INPUT
		Filter : REFERENCE TO exAssetIntUIFilterType;
	END_VAR
END_FUNCTION

FUNCTION exAssetIntCheckPreq : BOOL
	VAR_INPUT
		exLink : exAssetIntLinkType; (*Incoming communication handle (mapp standard interface)*) (* *) (*#PAR#;*)
		Logger : UDINT;
		State : REFERENCE TO exAssetIntStateEnum;
		StatusID : REFERENCE TO DINT;
		InfoDiagStatusID : REFERENCE TO exAssetIntStatusIDType;
	END_VAR
END_FUNCTION

FUNCTION exAssetIntCheckShiftData : BOOL
	VAR_INPUT
		Configuration : exAssetIntCoreConfigType;
		Logger : UDINT;
		State : REFERENCE TO exAssetIntStateEnum;
		StatusID : REFERENCE TO DINT;
		InfoDiagStatusID : REFERENCE TO exAssetIntStatusIDType;
	END_VAR
	VAR
		TmpStr1 : STRING[100];
		TmpStr2 : STRING[100];
		y : USINT;
		x : USINT;
	END_VAR
END_FUNCTION

FUNCTION InsertEventData : USINT
	VAR_INPUT
		Memory : UDINT;
		RecordCount : UINT;
		RecordData : exCoreInternalRecordType;
	END_VAR
	VAR
		RecordMemory : REFERENCE TO exCoreInternalRecordType;
		sort : UDINT;
		x : INT;
		y : INT;
	END_VAR
END_FUNCTION

FUNCTION CreateLoggerEntry : USINT
	VAR_INPUT
		LogLevel : exAssetIntLogLevelEnum; (*Log Level*)
		LogMsg : UDINT; (*Log message*)
		LogBuffer : UDINT; (*Address of log buffer*)
	END_VAR
	VAR
		RtcGettime : RTCtime_typ;
		TmpStr : STRING[20];
		LastMsg : STRING[LOG_LEN];
	END_VAR
END_FUNCTION

FUNCTION CreateErrorState : DINT
	VAR_INPUT
		ErrorID : DINT;
		ErrorMsg : UDINT; (*Log message*)
		Logger : UDINT;
		Severity : exComSeveritiesEnum;
		State : REFERENCE TO exAssetIntStateEnum;
		DiagStatusID : REFERENCE TO exAssetIntStatusIDType;
	END_VAR
END_FUNCTION

FUNCTION CalcStatsJob : USINT
	VAR_INPUT
		exLink : exAssetIntLinkType; (*Incoming communication handle (mapp standard interface)*) (* *) (*#PAR#;*)
		DiffLastCall : UDINT;
		Downtime : exAssetIntDowntimeEnum;
		Parameter : exAssetIntParType; (*Log Level*)
		JobStatistics : REFERENCE TO exAssetIntJobStatisticsType; (*Log message*)
	END_VAR
	VAR
		JobTotalTime : UDINT;
		Uptime : UDINT; (*Uptime in seconds*)
		NominalProductionTime : UDINT;
		GoodProductionTime : UDINT;
	END_VAR
END_FUNCTION

FUNCTION CalcStatsShift : USINT
	VAR_INPUT
		exLink : exAssetIntLinkType; (*Incoming communication handle (mapp standard interface)*) (* *) (*#PAR#;*)
		DiffLastCall : UDINT;
		Downtime : exAssetIntDowntimeEnum;
		Parameter : exAssetIntParType; (*Log Level*)
		ShiftStatistics : REFERENCE TO exAssetIntShiftStatisticsType; (*Log message*)
	END_VAR
	VAR
		ShiftTotalTime : UDINT;
		Uptime : UDINT; (*Uptime in seconds*)
		NominalProductionTime : UDINT;
		GoodProductionTime : UDINT;
	END_VAR
END_FUNCTION

FUNCTION CalcCrc : USINT
	VAR_INPUT
		data : UDINT;
		length : UINT;
	END_VAR
	VAR
		idx : UINT;
		_byte : USINT;
	END_VAR
END_FUNCTION

FUNCTION FindInstr : UDINT
	VAR_INPUT
		string1 : UDINT;
		string2 : UDINT;
	END_VAR
	VAR
		idx : UDINT;
	END_VAR
END_FUNCTION

FUNCTION ReplaceString : USINT
	VAR_INPUT
		dataSTR : UDINT;
		searchSTR : UDINT;
		replaceSTR : UDINT;
	END_VAR
	VAR
		idx : UDINT;
	END_VAR
END_FUNCTION

FUNCTION ReplaceDateTime : USINT
	VAR_INPUT
		dataSTR : UDINT;
		searchSTR : UDINT;
		value : UINT;
	END_VAR
	VAR
		lrealStr : LREAL;
	END_VAR
END_FUNCTION

FUNCTION NormalizeDateTime : LREAL
	VAR_INPUT
		value : UDINT;
	END_VAR
	VAR
		TmpStr1 : STRING[6] := '';
		TmpStr2 : STRING[6] := '';
	END_VAR
END_FUNCTION

FUNCTION NormalizeFloat : LREAL
	VAR_INPUT
		value : REAL;
		output : UDINT;
		configuration : exAssetIntExportType;
	END_VAR
	VAR
		idx : UDINT;
		tmpStr : STRING[50];
	END_VAR
END_FUNCTION
```
